// TIA Portal V17 export
// export: Created 2025-03-07T09:23:44.7208166Z, ExportSetting WithDefaults, DisplayName Totally Integrated Automation Portal, DisplayVersion V17 Update 8, DisplayName TIA Portal Openness, DisplayVersion V17 Update 8, DisplayName TIA Portal Version Control Interface, DisplayVersion V17, DisplayName SINAMICS Startdrive Advanced, DisplayVersion V17 SP2, DisplayName SINAMICS Startdrive G110M, G120, G120C, G120D, G120P, G115D, DisplayVersion V17 SP2, DisplayName SINAMICS Startdrive G130, G150, S120, S150, SINAMICS MV, S210, DisplayVersion V17 SP2, DisplayName STEP 7 Professional, DisplayVersion V17 Update 8, DisplayName SINUMERIK ONE STEP 7 Toolbox, DisplayVersion V17 Update 12, DisplayName SINUMERIK 840D sl STEP 7 Toolbox, DisplayVersion V17 Update 12, DisplayName STEP 7 Safety, DisplayVersion V17 Update 6, DisplayName WinCC Advanced, DisplayVersion V17 Update 8
FUNCTION "FC7238_VARIABLES_PLC_CONNECTION" : Void   // FC7238, LAD
{ S7_Optimized_Access := 'TRUE' }
VERSION : 0.1
// stored: AutoNumber false, IsIECCheckEnabled false, SetENOAutomatically false, UDAEnableTagReadback false
   VAR_TEMP
      AUX : Bool;
   END_VAR
   VAR_TEMP   // added for the SCL form of the ladder/FBD networks
      _w1 : Bool;
   END_VAR
BEGIN

REGION Network 1: FEEDERS GAS CHANGE CONDITIONS
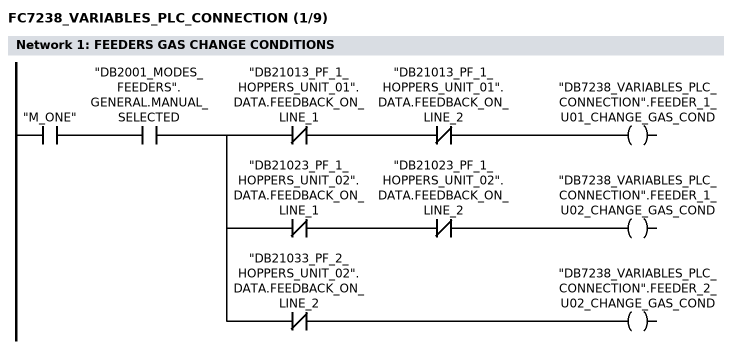
   RUNG wire#powerrail
      Contact( "M_ONE" )
      Contact( "DB2001_MODES_FEEDERS".GENERAL.MANUAL_SELECTED )
      wire#w1
      I_Contact( "DB21013_PF_1_HOPPERS_UNIT_01".DATA.FEEDBACK_ON_LINE_1 )
      I_Contact( "DB21013_PF_1_HOPPERS_UNIT_01".DATA.FEEDBACK_ON_LINE_2 )
      Coil( "DB7238_VARIABLES_PLC_CONNECTION".FEEDER_1_U01_CHANGE_GAS_COND )
   END_RUNG
   RUNG wire#w1
      I_Contact( "DB21023_PF_1_HOPPERS_UNIT_02".DATA.FEEDBACK_ON_LINE_1 )
      I_Contact( "DB21023_PF_1_HOPPERS_UNIT_02".DATA.FEEDBACK_ON_LINE_2 )
      Coil( "DB7238_VARIABLES_PLC_CONNECTION".FEEDER_1_U02_CHANGE_GAS_COND )
   END_RUNG
   RUNG wire#w1
      I_Contact( "DB21033_PF_2_HOPPERS_UNIT_02".DATA.FEEDBACK_ON_LINE_2 )
      Coil( "DB7238_VARIABLES_PLC_CONNECTION".FEEDER_2_U02_CHANGE_GAS_COND )
   END_RUNG
   // the same network as SCL:
   #_w1 := "M_ONE" AND "DB2001_MODES_FEEDERS".GENERAL.MANUAL_SELECTED;
   "DB7238_VARIABLES_PLC_CONNECTION".FEEDER_1_U01_CHANGE_GAS_COND := #_w1 AND NOT "DB21013_PF_1_HOPPERS_UNIT_01".DATA.FEEDBACK_ON_LINE_1 AND NOT "DB21013_PF_1_HOPPERS_UNIT_01".DATA.FEEDBACK_ON_LINE_2;
   "DB7238_VARIABLES_PLC_CONNECTION".FEEDER_1_U02_CHANGE_GAS_COND := #_w1 AND NOT "DB21023_PF_1_HOPPERS_UNIT_02".DATA.FEEDBACK_ON_LINE_1 AND NOT "DB21023_PF_1_HOPPERS_UNIT_02".DATA.FEEDBACK_ON_LINE_2;
   "DB7238_VARIABLES_PLC_CONNECTION".FEEDER_2_U02_CHANGE_GAS_COND := #_w1 AND NOT "DB21033_PF_2_HOPPERS_UNIT_02".DATA.FEEDBACK_ON_LINE_2;
END_REGION

REGION Network 2: FEEDER 1 UNIT 01 LINE 1
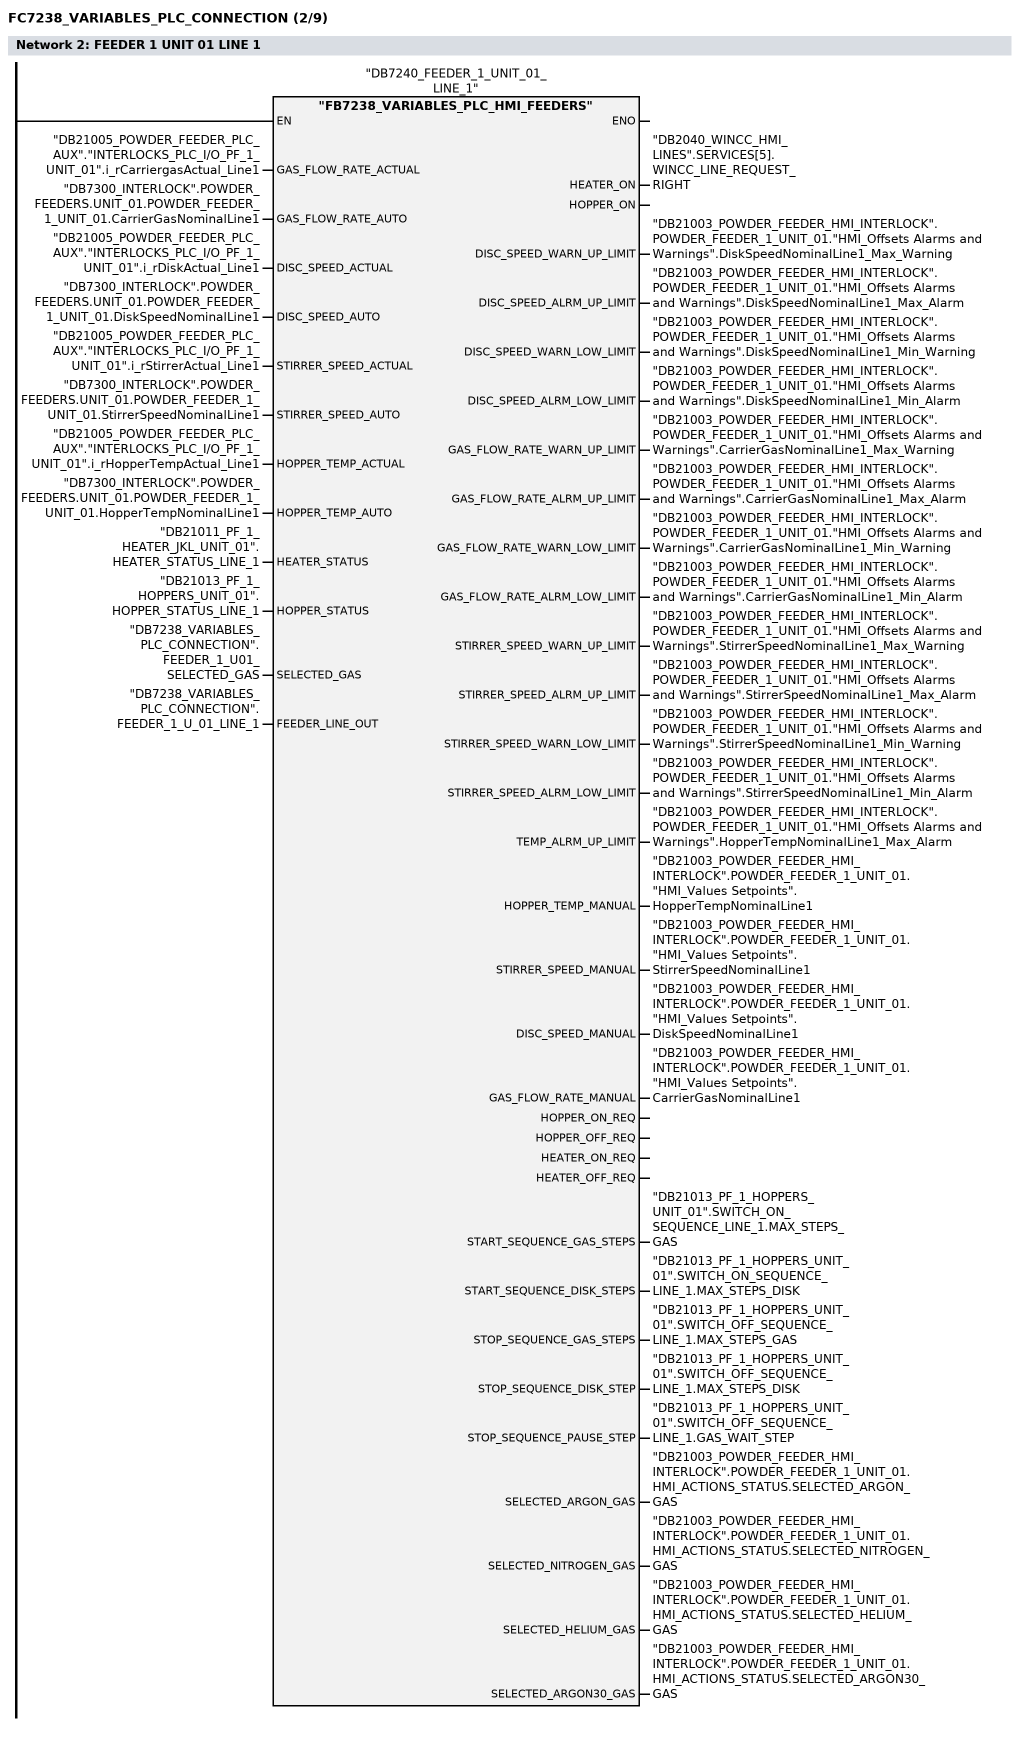
   RUNG wire#powerrail
      "DB7240_FEEDER_1_UNIT_01_LINE_1"(GAS_FLOW_RATE_ACTUAL := "DB21005_POWDER_FEEDER_PLC_AUX"."INTERLOCKS_PLC_I/O_PF_1_UNIT_01".i_rCarriergasActual_Line1, GAS_FLOW_RATE_AUTO := "DB7300_INTERLOCK".POWDER_FEEDERS.UNIT_01.POWDER_FEEDER_1_UNIT_01.CarrierGasNominalLine1, DISC_SPEED_ACTUAL := "DB21005_POWDER_FEEDER_PLC_AUX"."INTERLOCKS_PLC_I/O_PF_1_UNIT_01".i_rDiskActual_Line1, DISC_SPEED_AUTO := "DB7300_INTERLOCK".POWDER_FEEDERS.UNIT_01.POWDER_FEEDER_1_UNIT_01.DiskSpeedNominalLine1, STIRRER_SPEED_ACTUAL := "DB21005_POWDER_FEEDER_PLC_AUX"."INTERLOCKS_PLC_I/O_PF_1_UNIT_01".i_rStirrerActual_Line1, STIRRER_SPEED_AUTO := "DB7300_INTERLOCK".POWDER_FEEDERS.UNIT_01.POWDER_FEEDER_1_UNIT_01.StirrerSpeedNominalLine1, HOPPER_TEMP_ACTUAL := "DB21005_POWDER_FEEDER_PLC_AUX"."INTERLOCKS_PLC_I/O_PF_1_UNIT_01".i_rHopperTempActual_Line1, HOPPER_TEMP_AUTO := "DB7300_INTERLOCK".POWDER_FEEDERS.UNIT_01.POWDER_FEEDER_1_UNIT_01.HopperTempNominalLine1, HEATER_STATUS := "DB21011_PF_1_HEATER_JKL_UNIT_01".HEATER_STATUS_LINE_1, HOPPER_STATUS := "DB21013_PF_1_HOPPERS_UNIT_01".HOPPER_STATUS_LINE_1, SELECTED_GAS := "DB7238_VARIABLES_PLC_CONNECTION".FEEDER_1_U01_SELECTED_GAS, FEEDER_LINE_OUT := "DB7238_VARIABLES_PLC_CONNECTION".FEEDER_1_U_01_LINE_1, HEATER_ON => "DB2040_WINCC_HMI_LINES".SERVICES[5].WINCC_LINE_REQUEST_RIGHT, HOPPER_ON =>, DISC_SPEED_WARN_UP_LIMIT => "DB21003_POWDER_FEEDER_HMI_INTERLOCK".POWDER_FEEDER_1_UNIT_01."HMI_Offsets Alarms and Warnings".DiskSpeedNominalLine1_Max_Warning, DISC_SPEED_ALRM_UP_LIMIT => "DB21003_POWDER_FEEDER_HMI_INTERLOCK".POWDER_FEEDER_1_UNIT_01."HMI_Offsets Alarms and Warnings".DiskSpeedNominalLine1_Max_Alarm, DISC_SPEED_WARN_LOW_LIMIT => "DB21003_POWDER_FEEDER_HMI_INTERLOCK".POWDER_FEEDER_1_UNIT_01."HMI_Offsets Alarms and Warnings".DiskSpeedNominalLine1_Min_Warning, DISC_SPEED_ALRM_LOW_LIMIT => "DB21003_POWDER_FEEDER_HMI_INTERLOCK".POWDER_FEEDER_1_UNIT_01."HMI_Offsets Alarms and Warnings".DiskSpeedNominalLine1_Min_Alarm, GAS_FLOW_RATE_WARN_UP_LIMIT => "DB21003_POWDER_FEEDER_HMI_INTERLOCK".POWDER_FEEDER_1_UNIT_01."HMI_Offsets Alarms and Warnings".CarrierGasNominalLine1_Max_Warning, GAS_FLOW_RATE_ALRM_UP_LIMIT => "DB21003_POWDER_FEEDER_HMI_INTERLOCK".POWDER_FEEDER_1_UNIT_01."HMI_Offsets Alarms and Warnings".CarrierGasNominalLine1_Max_Alarm, GAS_FLOW_RATE_WARN_LOW_LIMIT => "DB21003_POWDER_FEEDER_HMI_INTERLOCK".POWDER_FEEDER_1_UNIT_01."HMI_Offsets Alarms and Warnings".CarrierGasNominalLine1_Min_Warning, GAS_FLOW_RATE_ALRM_LOW_LIMIT => "DB21003_POWDER_FEEDER_HMI_INTERLOCK".POWDER_FEEDER_1_UNIT_01."HMI_Offsets Alarms and Warnings".CarrierGasNominalLine1_Min_Alarm, STIRRER_SPEED_WARN_UP_LIMIT => "DB21003_POWDER_FEEDER_HMI_INTERLOCK".POWDER_FEEDER_1_UNIT_01."HMI_Offsets Alarms and Warnings".StirrerSpeedNominalLine1_Max_Warning, STIRRER_SPEED_ALRM_UP_LIMIT => "DB21003_POWDER_FEEDER_HMI_INTERLOCK".POWDER_FEEDER_1_UNIT_01."HMI_Offsets Alarms and Warnings".StirrerSpeedNominalLine1_Max_Alarm, STIRRER_SPEED_WARN_LOW_LIMIT => "DB21003_POWDER_FEEDER_HMI_INTERLOCK".POWDER_FEEDER_1_UNIT_01."HMI_Offsets Alarms and Warnings".StirrerSpeedNominalLine1_Min_Warning, STIRRER_SPEED_ALRM_LOW_LIMIT => "DB21003_POWDER_FEEDER_HMI_INTERLOCK".POWDER_FEEDER_1_UNIT_01."HMI_Offsets Alarms and Warnings".StirrerSpeedNominalLine1_Min_Alarm, TEMP_ALRM_UP_LIMIT => "DB21003_POWDER_FEEDER_HMI_INTERLOCK".POWDER_FEEDER_1_UNIT_01."HMI_Offsets Alarms and Warnings".HopperTempNominalLine1_Max_Alarm, HOPPER_TEMP_MANUAL => "DB21003_POWDER_FEEDER_HMI_INTERLOCK".POWDER_FEEDER_1_UNIT_01."HMI_Values Setpoints".HopperTempNominalLine1, STIRRER_SPEED_MANUAL => "DB21003_POWDER_FEEDER_HMI_INTERLOCK".POWDER_FEEDER_1_UNIT_01."HMI_Values Setpoints".StirrerSpeedNominalLine1, DISC_SPEED_MANUAL => "DB21003_POWDER_FEEDER_HMI_INTERLOCK".POWDER_FEEDER_1_UNIT_01."HMI_Values Setpoints".DiskSpeedNominalLine1, GAS_FLOW_RATE_MANUAL => "DB21003_POWDER_FEEDER_HMI_INTERLOCK".POWDER_FEEDER_1_UNIT_01."HMI_Values Setpoints".CarrierGasNominalLine1, HOPPER_ON_REQ =>, HOPPER_OFF_REQ =>, HEATER_ON_REQ =>, HEATER_OFF_REQ =>, START_SEQUENCE_GAS_STEPS => "DB21013_PF_1_HOPPERS_UNIT_01".SWITCH_ON_SEQUENCE_LINE_1.MAX_STEPS_GAS, START_SEQUENCE_DISK_STEPS => "DB21013_PF_1_HOPPERS_UNIT_01".SWITCH_ON_SEQUENCE_LINE_1.MAX_STEPS_DISK, STOP_SEQUENCE_GAS_STEPS => "DB21013_PF_1_HOPPERS_UNIT_01".SWITCH_OFF_SEQUENCE_LINE_1.MAX_STEPS_GAS, STOP_SEQUENCE_DISK_STEP => "DB21013_PF_1_HOPPERS_UNIT_01".SWITCH_OFF_SEQUENCE_LINE_1.MAX_STEPS_DISK, STOP_SEQUENCE_PAUSE_STEP => "DB21013_PF_1_HOPPERS_UNIT_01".SWITCH_OFF_SEQUENCE_LINE_1.GAS_WAIT_STEP, SELECTED_ARGON_GAS => "DB21003_POWDER_FEEDER_HMI_INTERLOCK".POWDER_FEEDER_1_UNIT_01.HMI_ACTIONS_STATUS.SELECTED_ARGON_GAS, SELECTED_NITROGEN_GAS => "DB21003_POWDER_FEEDER_HMI_INTERLOCK".POWDER_FEEDER_1_UNIT_01.HMI_ACTIONS_STATUS.SELECTED_NITROGEN_GAS, SELECTED_HELIUM_GAS => "DB21003_POWDER_FEEDER_HMI_INTERLOCK".POWDER_FEEDER_1_UNIT_01.HMI_ACTIONS_STATUS.SELECTED_HELIUM_GAS, SELECTED_ARGON30_GAS => "DB21003_POWDER_FEEDER_HMI_INTERLOCK".POWDER_FEEDER_1_UNIT_01.HMI_ACTIONS_STATUS.SELECTED_ARGON30_GAS)
   END_RUNG
   // the same network as SCL:
   "DB7240_FEEDER_1_UNIT_01_LINE_1"(GAS_FLOW_RATE_ACTUAL := "DB21005_POWDER_FEEDER_PLC_AUX"."INTERLOCKS_PLC_I/O_PF_1_UNIT_01".i_rCarriergasActual_Line1,   // "FB7238_VARIABLES_PLC_HMI_FEEDERS"
                           GAS_FLOW_RATE_AUTO := "DB7300_INTERLOCK".POWDER_FEEDERS.UNIT_01.POWDER_FEEDER_1_UNIT_01.CarrierGasNominalLine1,
                           DISC_SPEED_ACTUAL := "DB21005_POWDER_FEEDER_PLC_AUX"."INTERLOCKS_PLC_I/O_PF_1_UNIT_01".i_rDiskActual_Line1,
                           DISC_SPEED_AUTO := "DB7300_INTERLOCK".POWDER_FEEDERS.UNIT_01.POWDER_FEEDER_1_UNIT_01.DiskSpeedNominalLine1,
                           STIRRER_SPEED_ACTUAL := "DB21005_POWDER_FEEDER_PLC_AUX"."INTERLOCKS_PLC_I/O_PF_1_UNIT_01".i_rStirrerActual_Line1,
                           STIRRER_SPEED_AUTO := "DB7300_INTERLOCK".POWDER_FEEDERS.UNIT_01.POWDER_FEEDER_1_UNIT_01.StirrerSpeedNominalLine1,
                           HOPPER_TEMP_ACTUAL := "DB21005_POWDER_FEEDER_PLC_AUX"."INTERLOCKS_PLC_I/O_PF_1_UNIT_01".i_rHopperTempActual_Line1,
                           HOPPER_TEMP_AUTO := "DB7300_INTERLOCK".POWDER_FEEDERS.UNIT_01.POWDER_FEEDER_1_UNIT_01.HopperTempNominalLine1,
                           HEATER_STATUS := "DB21011_PF_1_HEATER_JKL_UNIT_01".HEATER_STATUS_LINE_1,
                           HOPPER_STATUS := "DB21013_PF_1_HOPPERS_UNIT_01".HOPPER_STATUS_LINE_1,
                           SELECTED_GAS := "DB7238_VARIABLES_PLC_CONNECTION".FEEDER_1_U01_SELECTED_GAS,
                           FEEDER_LINE_OUT := "DB7238_VARIABLES_PLC_CONNECTION".FEEDER_1_U_01_LINE_1,
                           HEATER_ON => "DB2040_WINCC_HMI_LINES".SERVICES[5].WINCC_LINE_REQUEST_RIGHT,
                           DISC_SPEED_WARN_UP_LIMIT => "DB21003_POWDER_FEEDER_HMI_INTERLOCK".POWDER_FEEDER_1_UNIT_01."HMI_Offsets Alarms and Warnings".DiskSpeedNominalLine1_Max_Warning,
                           DISC_SPEED_ALRM_UP_LIMIT => "DB21003_POWDER_FEEDER_HMI_INTERLOCK".POWDER_FEEDER_1_UNIT_01."HMI_Offsets Alarms and Warnings".DiskSpeedNominalLine1_Max_Alarm,
                           DISC_SPEED_WARN_LOW_LIMIT => "DB21003_POWDER_FEEDER_HMI_INTERLOCK".POWDER_FEEDER_1_UNIT_01."HMI_Offsets Alarms and Warnings".DiskSpeedNominalLine1_Min_Warning,
                           DISC_SPEED_ALRM_LOW_LIMIT => "DB21003_POWDER_FEEDER_HMI_INTERLOCK".POWDER_FEEDER_1_UNIT_01."HMI_Offsets Alarms and Warnings".DiskSpeedNominalLine1_Min_Alarm,
                           GAS_FLOW_RATE_WARN_UP_LIMIT => "DB21003_POWDER_FEEDER_HMI_INTERLOCK".POWDER_FEEDER_1_UNIT_01."HMI_Offsets Alarms and Warnings".CarrierGasNominalLine1_Max_Warning,
                           GAS_FLOW_RATE_ALRM_UP_LIMIT => "DB21003_POWDER_FEEDER_HMI_INTERLOCK".POWDER_FEEDER_1_UNIT_01."HMI_Offsets Alarms and Warnings".CarrierGasNominalLine1_Max_Alarm,
                           GAS_FLOW_RATE_WARN_LOW_LIMIT => "DB21003_POWDER_FEEDER_HMI_INTERLOCK".POWDER_FEEDER_1_UNIT_01."HMI_Offsets Alarms and Warnings".CarrierGasNominalLine1_Min_Warning,
                           GAS_FLOW_RATE_ALRM_LOW_LIMIT => "DB21003_POWDER_FEEDER_HMI_INTERLOCK".POWDER_FEEDER_1_UNIT_01."HMI_Offsets Alarms and Warnings".CarrierGasNominalLine1_Min_Alarm,
                           STIRRER_SPEED_WARN_UP_LIMIT => "DB21003_POWDER_FEEDER_HMI_INTERLOCK".POWDER_FEEDER_1_UNIT_01."HMI_Offsets Alarms and Warnings".StirrerSpeedNominalLine1_Max_Warning,
                           STIRRER_SPEED_ALRM_UP_LIMIT => "DB21003_POWDER_FEEDER_HMI_INTERLOCK".POWDER_FEEDER_1_UNIT_01."HMI_Offsets Alarms and Warnings".StirrerSpeedNominalLine1_Max_Alarm,
                           STIRRER_SPEED_WARN_LOW_LIMIT => "DB21003_POWDER_FEEDER_HMI_INTERLOCK".POWDER_FEEDER_1_UNIT_01."HMI_Offsets Alarms and Warnings".StirrerSpeedNominalLine1_Min_Warning,
                           STIRRER_SPEED_ALRM_LOW_LIMIT => "DB21003_POWDER_FEEDER_HMI_INTERLOCK".POWDER_FEEDER_1_UNIT_01."HMI_Offsets Alarms and Warnings".StirrerSpeedNominalLine1_Min_Alarm,
                           TEMP_ALRM_UP_LIMIT => "DB21003_POWDER_FEEDER_HMI_INTERLOCK".POWDER_FEEDER_1_UNIT_01."HMI_Offsets Alarms and Warnings".HopperTempNominalLine1_Max_Alarm,
                           HOPPER_TEMP_MANUAL => "DB21003_POWDER_FEEDER_HMI_INTERLOCK".POWDER_FEEDER_1_UNIT_01."HMI_Values Setpoints".HopperTempNominalLine1,
                           STIRRER_SPEED_MANUAL => "DB21003_POWDER_FEEDER_HMI_INTERLOCK".POWDER_FEEDER_1_UNIT_01."HMI_Values Setpoints".StirrerSpeedNominalLine1,
                           DISC_SPEED_MANUAL => "DB21003_POWDER_FEEDER_HMI_INTERLOCK".POWDER_FEEDER_1_UNIT_01."HMI_Values Setpoints".DiskSpeedNominalLine1,
                           GAS_FLOW_RATE_MANUAL => "DB21003_POWDER_FEEDER_HMI_INTERLOCK".POWDER_FEEDER_1_UNIT_01."HMI_Values Setpoints".CarrierGasNominalLine1,
                           START_SEQUENCE_GAS_STEPS => "DB21013_PF_1_HOPPERS_UNIT_01".SWITCH_ON_SEQUENCE_LINE_1.MAX_STEPS_GAS,
                           START_SEQUENCE_DISK_STEPS => "DB21013_PF_1_HOPPERS_UNIT_01".SWITCH_ON_SEQUENCE_LINE_1.MAX_STEPS_DISK,
                           STOP_SEQUENCE_GAS_STEPS => "DB21013_PF_1_HOPPERS_UNIT_01".SWITCH_OFF_SEQUENCE_LINE_1.MAX_STEPS_GAS,
                           STOP_SEQUENCE_DISK_STEP => "DB21013_PF_1_HOPPERS_UNIT_01".SWITCH_OFF_SEQUENCE_LINE_1.MAX_STEPS_DISK,
                           STOP_SEQUENCE_PAUSE_STEP => "DB21013_PF_1_HOPPERS_UNIT_01".SWITCH_OFF_SEQUENCE_LINE_1.GAS_WAIT_STEP,
                           SELECTED_ARGON_GAS => "DB21003_POWDER_FEEDER_HMI_INTERLOCK".POWDER_FEEDER_1_UNIT_01.HMI_ACTIONS_STATUS.SELECTED_ARGON_GAS,
                           SELECTED_NITROGEN_GAS => "DB21003_POWDER_FEEDER_HMI_INTERLOCK".POWDER_FEEDER_1_UNIT_01.HMI_ACTIONS_STATUS.SELECTED_NITROGEN_GAS,
                           SELECTED_HELIUM_GAS => "DB21003_POWDER_FEEDER_HMI_INTERLOCK".POWDER_FEEDER_1_UNIT_01.HMI_ACTIONS_STATUS.SELECTED_HELIUM_GAS,
                           SELECTED_ARGON30_GAS => "DB21003_POWDER_FEEDER_HMI_INTERLOCK".POWDER_FEEDER_1_UNIT_01.HMI_ACTIONS_STATUS.SELECTED_ARGON30_GAS);
END_REGION

REGION Network 3: FEEDER 1 UNIT 01 LINE 2
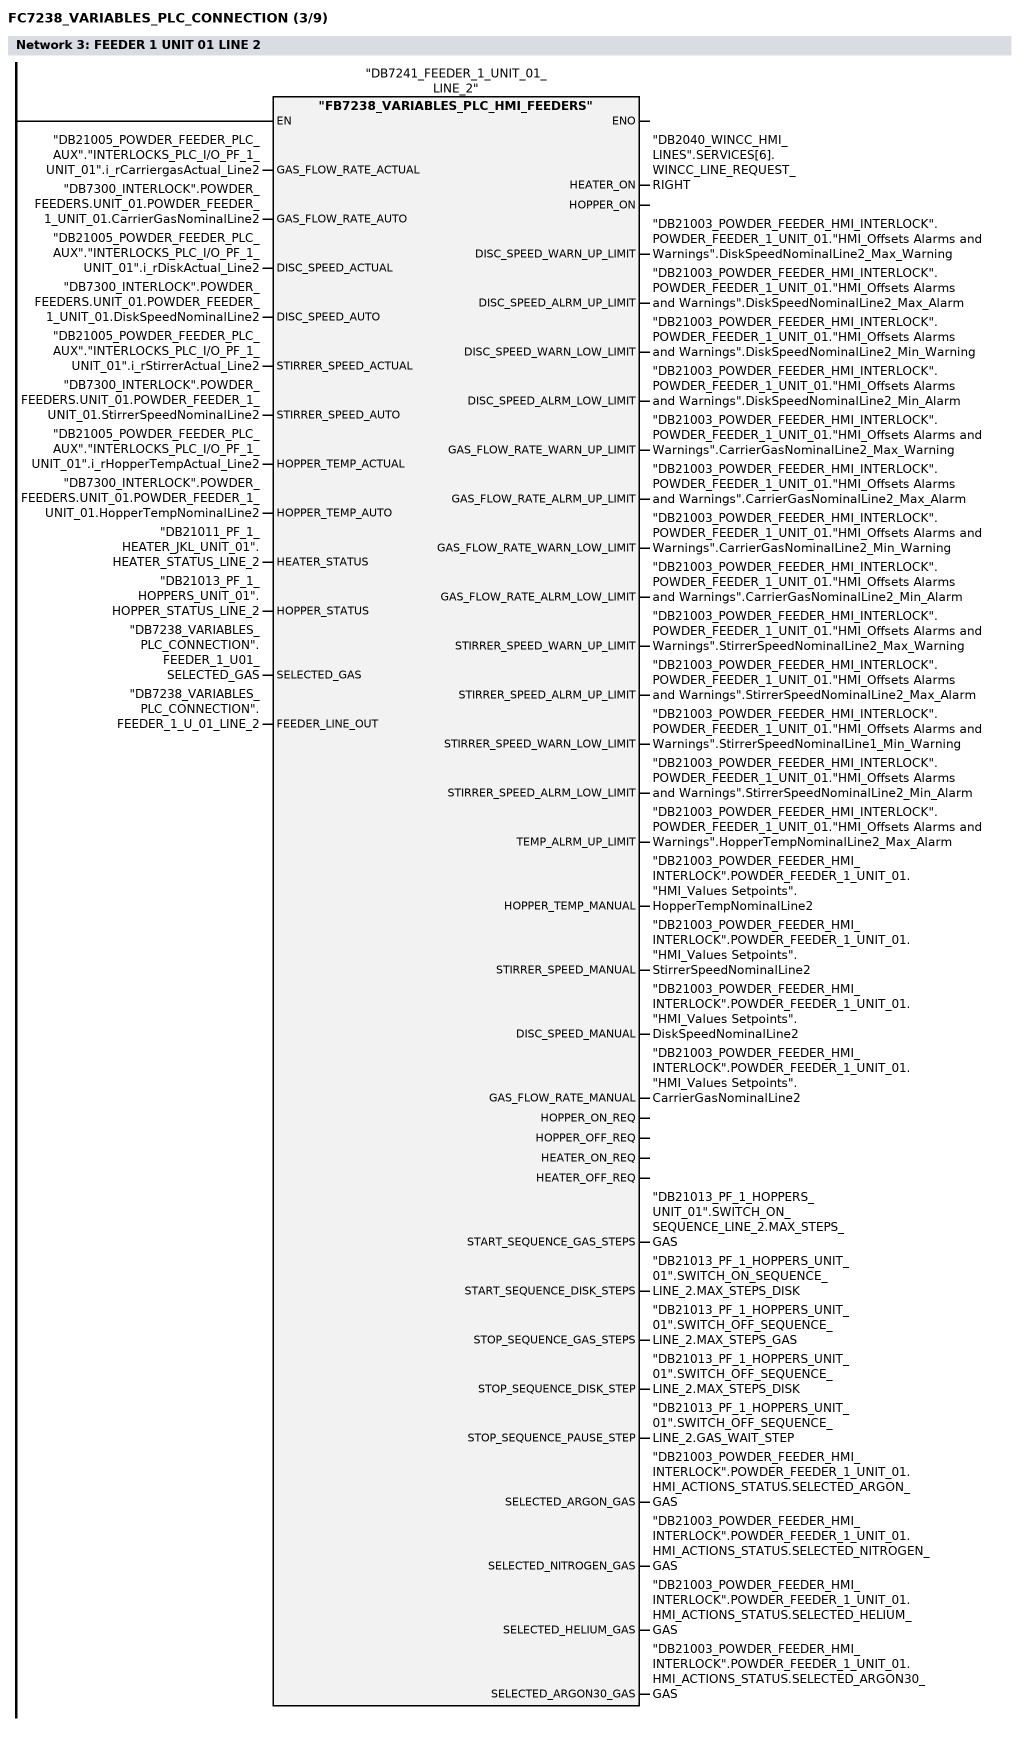
   RUNG wire#powerrail
      "DB7241_FEEDER_1_UNIT_01_LINE_2"(GAS_FLOW_RATE_ACTUAL := "DB21005_POWDER_FEEDER_PLC_AUX"."INTERLOCKS_PLC_I/O_PF_1_UNIT_01".i_rCarriergasActual_Line2, GAS_FLOW_RATE_AUTO := "DB7300_INTERLOCK".POWDER_FEEDERS.UNIT_01.POWDER_FEEDER_1_UNIT_01.CarrierGasNominalLine2, DISC_SPEED_ACTUAL := "DB21005_POWDER_FEEDER_PLC_AUX"."INTERLOCKS_PLC_I/O_PF_1_UNIT_01".i_rDiskActual_Line2, DISC_SPEED_AUTO := "DB7300_INTERLOCK".POWDER_FEEDERS.UNIT_01.POWDER_FEEDER_1_UNIT_01.DiskSpeedNominalLine2, STIRRER_SPEED_ACTUAL := "DB21005_POWDER_FEEDER_PLC_AUX"."INTERLOCKS_PLC_I/O_PF_1_UNIT_01".i_rStirrerActual_Line2, STIRRER_SPEED_AUTO := "DB7300_INTERLOCK".POWDER_FEEDERS.UNIT_01.POWDER_FEEDER_1_UNIT_01.StirrerSpeedNominalLine2, HOPPER_TEMP_ACTUAL := "DB21005_POWDER_FEEDER_PLC_AUX"."INTERLOCKS_PLC_I/O_PF_1_UNIT_01".i_rHopperTempActual_Line2, HOPPER_TEMP_AUTO := "DB7300_INTERLOCK".POWDER_FEEDERS.UNIT_01.POWDER_FEEDER_1_UNIT_01.HopperTempNominalLine2, HEATER_STATUS := "DB21011_PF_1_HEATER_JKL_UNIT_01".HEATER_STATUS_LINE_2, HOPPER_STATUS := "DB21013_PF_1_HOPPERS_UNIT_01".HOPPER_STATUS_LINE_2, SELECTED_GAS := "DB7238_VARIABLES_PLC_CONNECTION".FEEDER_1_U01_SELECTED_GAS, FEEDER_LINE_OUT := "DB7238_VARIABLES_PLC_CONNECTION".FEEDER_1_U_01_LINE_2, HEATER_ON => "DB2040_WINCC_HMI_LINES".SERVICES[6].WINCC_LINE_REQUEST_RIGHT, HOPPER_ON =>, DISC_SPEED_WARN_UP_LIMIT => "DB21003_POWDER_FEEDER_HMI_INTERLOCK".POWDER_FEEDER_1_UNIT_01."HMI_Offsets Alarms and Warnings".DiskSpeedNominalLine2_Max_Warning, DISC_SPEED_ALRM_UP_LIMIT => "DB21003_POWDER_FEEDER_HMI_INTERLOCK".POWDER_FEEDER_1_UNIT_01."HMI_Offsets Alarms and Warnings".DiskSpeedNominalLine2_Max_Alarm, DISC_SPEED_WARN_LOW_LIMIT => "DB21003_POWDER_FEEDER_HMI_INTERLOCK".POWDER_FEEDER_1_UNIT_01."HMI_Offsets Alarms and Warnings".DiskSpeedNominalLine2_Min_Warning, DISC_SPEED_ALRM_LOW_LIMIT => "DB21003_POWDER_FEEDER_HMI_INTERLOCK".POWDER_FEEDER_1_UNIT_01."HMI_Offsets Alarms and Warnings".DiskSpeedNominalLine2_Min_Alarm, GAS_FLOW_RATE_WARN_UP_LIMIT => "DB21003_POWDER_FEEDER_HMI_INTERLOCK".POWDER_FEEDER_1_UNIT_01."HMI_Offsets Alarms and Warnings".CarrierGasNominalLine2_Max_Warning, GAS_FLOW_RATE_ALRM_UP_LIMIT => "DB21003_POWDER_FEEDER_HMI_INTERLOCK".POWDER_FEEDER_1_UNIT_01."HMI_Offsets Alarms and Warnings".CarrierGasNominalLine2_Max_Alarm, GAS_FLOW_RATE_WARN_LOW_LIMIT => "DB21003_POWDER_FEEDER_HMI_INTERLOCK".POWDER_FEEDER_1_UNIT_01."HMI_Offsets Alarms and Warnings".CarrierGasNominalLine2_Min_Warning, GAS_FLOW_RATE_ALRM_LOW_LIMIT => "DB21003_POWDER_FEEDER_HMI_INTERLOCK".POWDER_FEEDER_1_UNIT_01."HMI_Offsets Alarms and Warnings".CarrierGasNominalLine2_Min_Alarm, STIRRER_SPEED_WARN_UP_LIMIT => "DB21003_POWDER_FEEDER_HMI_INTERLOCK".POWDER_FEEDER_1_UNIT_01."HMI_Offsets Alarms and Warnings".StirrerSpeedNominalLine2_Max_Warning, STIRRER_SPEED_ALRM_UP_LIMIT => "DB21003_POWDER_FEEDER_HMI_INTERLOCK".POWDER_FEEDER_1_UNIT_01."HMI_Offsets Alarms and Warnings".StirrerSpeedNominalLine2_Max_Alarm, STIRRER_SPEED_WARN_LOW_LIMIT => "DB21003_POWDER_FEEDER_HMI_INTERLOCK".POWDER_FEEDER_1_UNIT_01."HMI_Offsets Alarms and Warnings".StirrerSpeedNominalLine1_Min_Warning, STIRRER_SPEED_ALRM_LOW_LIMIT => "DB21003_POWDER_FEEDER_HMI_INTERLOCK".POWDER_FEEDER_1_UNIT_01."HMI_Offsets Alarms and Warnings".StirrerSpeedNominalLine2_Min_Alarm, TEMP_ALRM_UP_LIMIT => "DB21003_POWDER_FEEDER_HMI_INTERLOCK".POWDER_FEEDER_1_UNIT_01."HMI_Offsets Alarms and Warnings".HopperTempNominalLine2_Max_Alarm, HOPPER_TEMP_MANUAL => "DB21003_POWDER_FEEDER_HMI_INTERLOCK".POWDER_FEEDER_1_UNIT_01."HMI_Values Setpoints".HopperTempNominalLine2, STIRRER_SPEED_MANUAL => "DB21003_POWDER_FEEDER_HMI_INTERLOCK".POWDER_FEEDER_1_UNIT_01."HMI_Values Setpoints".StirrerSpeedNominalLine2, DISC_SPEED_MANUAL => "DB21003_POWDER_FEEDER_HMI_INTERLOCK".POWDER_FEEDER_1_UNIT_01."HMI_Values Setpoints".DiskSpeedNominalLine2, GAS_FLOW_RATE_MANUAL => "DB21003_POWDER_FEEDER_HMI_INTERLOCK".POWDER_FEEDER_1_UNIT_01."HMI_Values Setpoints".CarrierGasNominalLine2, HOPPER_ON_REQ =>, HOPPER_OFF_REQ =>, HEATER_ON_REQ =>, HEATER_OFF_REQ =>, START_SEQUENCE_GAS_STEPS => "DB21013_PF_1_HOPPERS_UNIT_01".SWITCH_ON_SEQUENCE_LINE_2.MAX_STEPS_GAS, START_SEQUENCE_DISK_STEPS => "DB21013_PF_1_HOPPERS_UNIT_01".SWITCH_ON_SEQUENCE_LINE_2.MAX_STEPS_DISK, STOP_SEQUENCE_GAS_STEPS => "DB21013_PF_1_HOPPERS_UNIT_01".SWITCH_OFF_SEQUENCE_LINE_2.MAX_STEPS_GAS, STOP_SEQUENCE_DISK_STEP => "DB21013_PF_1_HOPPERS_UNIT_01".SWITCH_OFF_SEQUENCE_LINE_2.MAX_STEPS_DISK, STOP_SEQUENCE_PAUSE_STEP => "DB21013_PF_1_HOPPERS_UNIT_01".SWITCH_OFF_SEQUENCE_LINE_2.GAS_WAIT_STEP, SELECTED_ARGON_GAS => "DB21003_POWDER_FEEDER_HMI_INTERLOCK".POWDER_FEEDER_1_UNIT_01.HMI_ACTIONS_STATUS.SELECTED_ARGON_GAS, SELECTED_NITROGEN_GAS => "DB21003_POWDER_FEEDER_HMI_INTERLOCK".POWDER_FEEDER_1_UNIT_01.HMI_ACTIONS_STATUS.SELECTED_NITROGEN_GAS, SELECTED_HELIUM_GAS => "DB21003_POWDER_FEEDER_HMI_INTERLOCK".POWDER_FEEDER_1_UNIT_01.HMI_ACTIONS_STATUS.SELECTED_HELIUM_GAS, SELECTED_ARGON30_GAS => "DB21003_POWDER_FEEDER_HMI_INTERLOCK".POWDER_FEEDER_1_UNIT_01.HMI_ACTIONS_STATUS.SELECTED_ARGON30_GAS)
   END_RUNG
   // the same network as SCL:
   "DB7241_FEEDER_1_UNIT_01_LINE_2"(GAS_FLOW_RATE_ACTUAL := "DB21005_POWDER_FEEDER_PLC_AUX"."INTERLOCKS_PLC_I/O_PF_1_UNIT_01".i_rCarriergasActual_Line2,   // "FB7238_VARIABLES_PLC_HMI_FEEDERS"
                           GAS_FLOW_RATE_AUTO := "DB7300_INTERLOCK".POWDER_FEEDERS.UNIT_01.POWDER_FEEDER_1_UNIT_01.CarrierGasNominalLine2,
                           DISC_SPEED_ACTUAL := "DB21005_POWDER_FEEDER_PLC_AUX"."INTERLOCKS_PLC_I/O_PF_1_UNIT_01".i_rDiskActual_Line2,
                           DISC_SPEED_AUTO := "DB7300_INTERLOCK".POWDER_FEEDERS.UNIT_01.POWDER_FEEDER_1_UNIT_01.DiskSpeedNominalLine2,
                           STIRRER_SPEED_ACTUAL := "DB21005_POWDER_FEEDER_PLC_AUX"."INTERLOCKS_PLC_I/O_PF_1_UNIT_01".i_rStirrerActual_Line2,
                           STIRRER_SPEED_AUTO := "DB7300_INTERLOCK".POWDER_FEEDERS.UNIT_01.POWDER_FEEDER_1_UNIT_01.StirrerSpeedNominalLine2,
                           HOPPER_TEMP_ACTUAL := "DB21005_POWDER_FEEDER_PLC_AUX"."INTERLOCKS_PLC_I/O_PF_1_UNIT_01".i_rHopperTempActual_Line2,
                           HOPPER_TEMP_AUTO := "DB7300_INTERLOCK".POWDER_FEEDERS.UNIT_01.POWDER_FEEDER_1_UNIT_01.HopperTempNominalLine2,
                           HEATER_STATUS := "DB21011_PF_1_HEATER_JKL_UNIT_01".HEATER_STATUS_LINE_2,
                           HOPPER_STATUS := "DB21013_PF_1_HOPPERS_UNIT_01".HOPPER_STATUS_LINE_2,
                           SELECTED_GAS := "DB7238_VARIABLES_PLC_CONNECTION".FEEDER_1_U01_SELECTED_GAS,
                           FEEDER_LINE_OUT := "DB7238_VARIABLES_PLC_CONNECTION".FEEDER_1_U_01_LINE_2,
                           HEATER_ON => "DB2040_WINCC_HMI_LINES".SERVICES[6].WINCC_LINE_REQUEST_RIGHT,
                           DISC_SPEED_WARN_UP_LIMIT => "DB21003_POWDER_FEEDER_HMI_INTERLOCK".POWDER_FEEDER_1_UNIT_01."HMI_Offsets Alarms and Warnings".DiskSpeedNominalLine2_Max_Warning,
                           DISC_SPEED_ALRM_UP_LIMIT => "DB21003_POWDER_FEEDER_HMI_INTERLOCK".POWDER_FEEDER_1_UNIT_01."HMI_Offsets Alarms and Warnings".DiskSpeedNominalLine2_Max_Alarm,
                           DISC_SPEED_WARN_LOW_LIMIT => "DB21003_POWDER_FEEDER_HMI_INTERLOCK".POWDER_FEEDER_1_UNIT_01."HMI_Offsets Alarms and Warnings".DiskSpeedNominalLine2_Min_Warning,
                           DISC_SPEED_ALRM_LOW_LIMIT => "DB21003_POWDER_FEEDER_HMI_INTERLOCK".POWDER_FEEDER_1_UNIT_01."HMI_Offsets Alarms and Warnings".DiskSpeedNominalLine2_Min_Alarm,
                           GAS_FLOW_RATE_WARN_UP_LIMIT => "DB21003_POWDER_FEEDER_HMI_INTERLOCK".POWDER_FEEDER_1_UNIT_01."HMI_Offsets Alarms and Warnings".CarrierGasNominalLine2_Max_Warning,
                           GAS_FLOW_RATE_ALRM_UP_LIMIT => "DB21003_POWDER_FEEDER_HMI_INTERLOCK".POWDER_FEEDER_1_UNIT_01."HMI_Offsets Alarms and Warnings".CarrierGasNominalLine2_Max_Alarm,
                           GAS_FLOW_RATE_WARN_LOW_LIMIT => "DB21003_POWDER_FEEDER_HMI_INTERLOCK".POWDER_FEEDER_1_UNIT_01."HMI_Offsets Alarms and Warnings".CarrierGasNominalLine2_Min_Warning,
                           GAS_FLOW_RATE_ALRM_LOW_LIMIT => "DB21003_POWDER_FEEDER_HMI_INTERLOCK".POWDER_FEEDER_1_UNIT_01."HMI_Offsets Alarms and Warnings".CarrierGasNominalLine2_Min_Alarm,
                           STIRRER_SPEED_WARN_UP_LIMIT => "DB21003_POWDER_FEEDER_HMI_INTERLOCK".POWDER_FEEDER_1_UNIT_01."HMI_Offsets Alarms and Warnings".StirrerSpeedNominalLine2_Max_Warning,
                           STIRRER_SPEED_ALRM_UP_LIMIT => "DB21003_POWDER_FEEDER_HMI_INTERLOCK".POWDER_FEEDER_1_UNIT_01."HMI_Offsets Alarms and Warnings".StirrerSpeedNominalLine2_Max_Alarm,
                           STIRRER_SPEED_WARN_LOW_LIMIT => "DB21003_POWDER_FEEDER_HMI_INTERLOCK".POWDER_FEEDER_1_UNIT_01."HMI_Offsets Alarms and Warnings".StirrerSpeedNominalLine1_Min_Warning,
                           STIRRER_SPEED_ALRM_LOW_LIMIT => "DB21003_POWDER_FEEDER_HMI_INTERLOCK".POWDER_FEEDER_1_UNIT_01."HMI_Offsets Alarms and Warnings".StirrerSpeedNominalLine2_Min_Alarm,
                           TEMP_ALRM_UP_LIMIT => "DB21003_POWDER_FEEDER_HMI_INTERLOCK".POWDER_FEEDER_1_UNIT_01."HMI_Offsets Alarms and Warnings".HopperTempNominalLine2_Max_Alarm,
                           HOPPER_TEMP_MANUAL => "DB21003_POWDER_FEEDER_HMI_INTERLOCK".POWDER_FEEDER_1_UNIT_01."HMI_Values Setpoints".HopperTempNominalLine2,
                           STIRRER_SPEED_MANUAL => "DB21003_POWDER_FEEDER_HMI_INTERLOCK".POWDER_FEEDER_1_UNIT_01."HMI_Values Setpoints".StirrerSpeedNominalLine2,
                           DISC_SPEED_MANUAL => "DB21003_POWDER_FEEDER_HMI_INTERLOCK".POWDER_FEEDER_1_UNIT_01."HMI_Values Setpoints".DiskSpeedNominalLine2,
                           GAS_FLOW_RATE_MANUAL => "DB21003_POWDER_FEEDER_HMI_INTERLOCK".POWDER_FEEDER_1_UNIT_01."HMI_Values Setpoints".CarrierGasNominalLine2,
                           START_SEQUENCE_GAS_STEPS => "DB21013_PF_1_HOPPERS_UNIT_01".SWITCH_ON_SEQUENCE_LINE_2.MAX_STEPS_GAS,
                           START_SEQUENCE_DISK_STEPS => "DB21013_PF_1_HOPPERS_UNIT_01".SWITCH_ON_SEQUENCE_LINE_2.MAX_STEPS_DISK,
                           STOP_SEQUENCE_GAS_STEPS => "DB21013_PF_1_HOPPERS_UNIT_01".SWITCH_OFF_SEQUENCE_LINE_2.MAX_STEPS_GAS,
                           STOP_SEQUENCE_DISK_STEP => "DB21013_PF_1_HOPPERS_UNIT_01".SWITCH_OFF_SEQUENCE_LINE_2.MAX_STEPS_DISK,
                           STOP_SEQUENCE_PAUSE_STEP => "DB21013_PF_1_HOPPERS_UNIT_01".SWITCH_OFF_SEQUENCE_LINE_2.GAS_WAIT_STEP,
                           SELECTED_ARGON_GAS => "DB21003_POWDER_FEEDER_HMI_INTERLOCK".POWDER_FEEDER_1_UNIT_01.HMI_ACTIONS_STATUS.SELECTED_ARGON_GAS,
                           SELECTED_NITROGEN_GAS => "DB21003_POWDER_FEEDER_HMI_INTERLOCK".POWDER_FEEDER_1_UNIT_01.HMI_ACTIONS_STATUS.SELECTED_NITROGEN_GAS,
                           SELECTED_HELIUM_GAS => "DB21003_POWDER_FEEDER_HMI_INTERLOCK".POWDER_FEEDER_1_UNIT_01.HMI_ACTIONS_STATUS.SELECTED_HELIUM_GAS,
                           SELECTED_ARGON30_GAS => "DB21003_POWDER_FEEDER_HMI_INTERLOCK".POWDER_FEEDER_1_UNIT_01.HMI_ACTIONS_STATUS.SELECTED_ARGON30_GAS);
END_REGION

REGION Network 4: FEEDER 1 UNIT 02 LINE 1
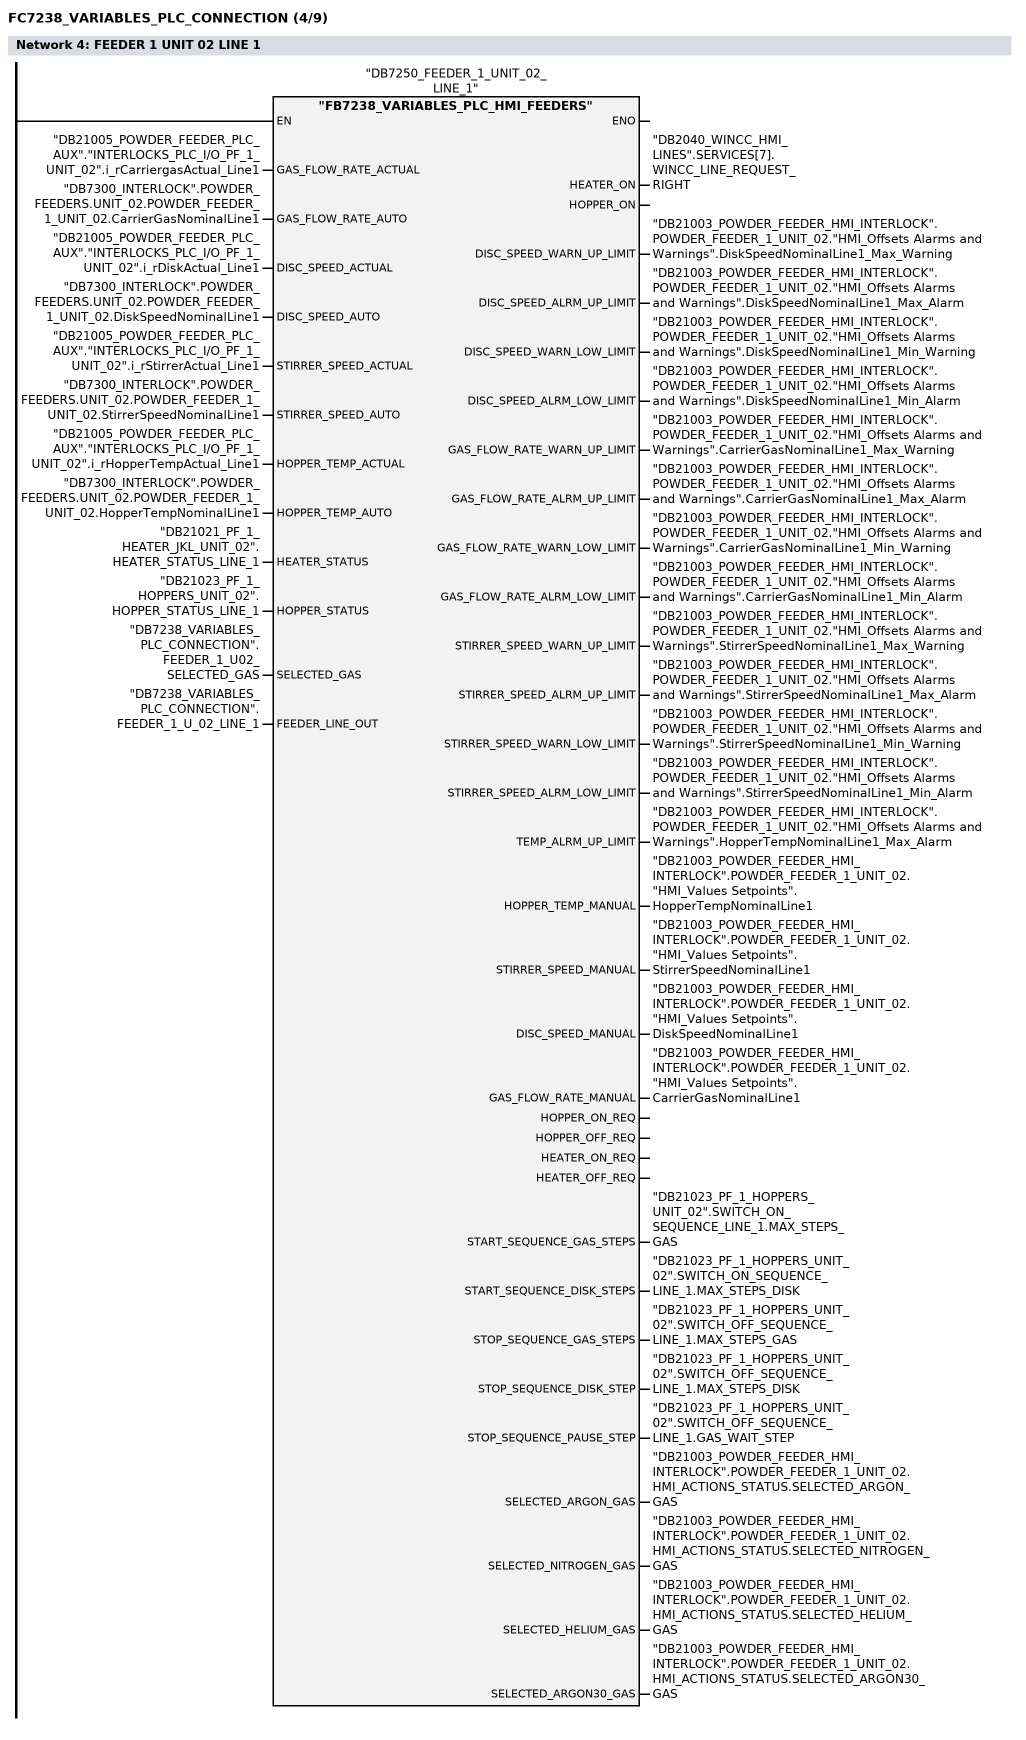
   RUNG wire#powerrail
      "DB7250_FEEDER_1_UNIT_02_LINE_1"(GAS_FLOW_RATE_ACTUAL := "DB21005_POWDER_FEEDER_PLC_AUX"."INTERLOCKS_PLC_I/O_PF_1_UNIT_02".i_rCarriergasActual_Line1, GAS_FLOW_RATE_AUTO := "DB7300_INTERLOCK".POWDER_FEEDERS.UNIT_02.POWDER_FEEDER_1_UNIT_02.CarrierGasNominalLine1, DISC_SPEED_ACTUAL := "DB21005_POWDER_FEEDER_PLC_AUX"."INTERLOCKS_PLC_I/O_PF_1_UNIT_02".i_rDiskActual_Line1, DISC_SPEED_AUTO := "DB7300_INTERLOCK".POWDER_FEEDERS.UNIT_02.POWDER_FEEDER_1_UNIT_02.DiskSpeedNominalLine1, STIRRER_SPEED_ACTUAL := "DB21005_POWDER_FEEDER_PLC_AUX"."INTERLOCKS_PLC_I/O_PF_1_UNIT_02".i_rStirrerActual_Line1, STIRRER_SPEED_AUTO := "DB7300_INTERLOCK".POWDER_FEEDERS.UNIT_02.POWDER_FEEDER_1_UNIT_02.StirrerSpeedNominalLine1, HOPPER_TEMP_ACTUAL := "DB21005_POWDER_FEEDER_PLC_AUX"."INTERLOCKS_PLC_I/O_PF_1_UNIT_02".i_rHopperTempActual_Line1, HOPPER_TEMP_AUTO := "DB7300_INTERLOCK".POWDER_FEEDERS.UNIT_02.POWDER_FEEDER_1_UNIT_02.HopperTempNominalLine1, HEATER_STATUS := "DB21021_PF_1_HEATER_JKL_UNIT_02".HEATER_STATUS_LINE_1, HOPPER_STATUS := "DB21023_PF_1_HOPPERS_UNIT_02".HOPPER_STATUS_LINE_1, SELECTED_GAS := "DB7238_VARIABLES_PLC_CONNECTION".FEEDER_1_U02_SELECTED_GAS, FEEDER_LINE_OUT := "DB7238_VARIABLES_PLC_CONNECTION".FEEDER_1_U_02_LINE_1, HEATER_ON => "DB2040_WINCC_HMI_LINES".SERVICES[7].WINCC_LINE_REQUEST_RIGHT, HOPPER_ON =>, DISC_SPEED_WARN_UP_LIMIT => "DB21003_POWDER_FEEDER_HMI_INTERLOCK".POWDER_FEEDER_1_UNIT_02."HMI_Offsets Alarms and Warnings".DiskSpeedNominalLine1_Max_Warning, DISC_SPEED_ALRM_UP_LIMIT => "DB21003_POWDER_FEEDER_HMI_INTERLOCK".POWDER_FEEDER_1_UNIT_02."HMI_Offsets Alarms and Warnings".DiskSpeedNominalLine1_Max_Alarm, DISC_SPEED_WARN_LOW_LIMIT => "DB21003_POWDER_FEEDER_HMI_INTERLOCK".POWDER_FEEDER_1_UNIT_02."HMI_Offsets Alarms and Warnings".DiskSpeedNominalLine1_Min_Warning, DISC_SPEED_ALRM_LOW_LIMIT => "DB21003_POWDER_FEEDER_HMI_INTERLOCK".POWDER_FEEDER_1_UNIT_02."HMI_Offsets Alarms and Warnings".DiskSpeedNominalLine1_Min_Alarm, GAS_FLOW_RATE_WARN_UP_LIMIT => "DB21003_POWDER_FEEDER_HMI_INTERLOCK".POWDER_FEEDER_1_UNIT_02."HMI_Offsets Alarms and Warnings".CarrierGasNominalLine1_Max_Warning, GAS_FLOW_RATE_ALRM_UP_LIMIT => "DB21003_POWDER_FEEDER_HMI_INTERLOCK".POWDER_FEEDER_1_UNIT_02."HMI_Offsets Alarms and Warnings".CarrierGasNominalLine1_Max_Alarm, GAS_FLOW_RATE_WARN_LOW_LIMIT => "DB21003_POWDER_FEEDER_HMI_INTERLOCK".POWDER_FEEDER_1_UNIT_02."HMI_Offsets Alarms and Warnings".CarrierGasNominalLine1_Min_Warning, GAS_FLOW_RATE_ALRM_LOW_LIMIT => "DB21003_POWDER_FEEDER_HMI_INTERLOCK".POWDER_FEEDER_1_UNIT_02."HMI_Offsets Alarms and Warnings".CarrierGasNominalLine1_Min_Alarm, STIRRER_SPEED_WARN_UP_LIMIT => "DB21003_POWDER_FEEDER_HMI_INTERLOCK".POWDER_FEEDER_1_UNIT_02."HMI_Offsets Alarms and Warnings".StirrerSpeedNominalLine1_Max_Warning, STIRRER_SPEED_ALRM_UP_LIMIT => "DB21003_POWDER_FEEDER_HMI_INTERLOCK".POWDER_FEEDER_1_UNIT_02."HMI_Offsets Alarms and Warnings".StirrerSpeedNominalLine1_Max_Alarm, STIRRER_SPEED_WARN_LOW_LIMIT => "DB21003_POWDER_FEEDER_HMI_INTERLOCK".POWDER_FEEDER_1_UNIT_02."HMI_Offsets Alarms and Warnings".StirrerSpeedNominalLine1_Min_Warning, STIRRER_SPEED_ALRM_LOW_LIMIT => "DB21003_POWDER_FEEDER_HMI_INTERLOCK".POWDER_FEEDER_1_UNIT_02."HMI_Offsets Alarms and Warnings".StirrerSpeedNominalLine1_Min_Alarm, TEMP_ALRM_UP_LIMIT => "DB21003_POWDER_FEEDER_HMI_INTERLOCK".POWDER_FEEDER_1_UNIT_02."HMI_Offsets Alarms and Warnings".HopperTempNominalLine1_Max_Alarm, HOPPER_TEMP_MANUAL => "DB21003_POWDER_FEEDER_HMI_INTERLOCK".POWDER_FEEDER_1_UNIT_02."HMI_Values Setpoints".HopperTempNominalLine1, STIRRER_SPEED_MANUAL => "DB21003_POWDER_FEEDER_HMI_INTERLOCK".POWDER_FEEDER_1_UNIT_02."HMI_Values Setpoints".StirrerSpeedNominalLine1, DISC_SPEED_MANUAL => "DB21003_POWDER_FEEDER_HMI_INTERLOCK".POWDER_FEEDER_1_UNIT_02."HMI_Values Setpoints".DiskSpeedNominalLine1, GAS_FLOW_RATE_MANUAL => "DB21003_POWDER_FEEDER_HMI_INTERLOCK".POWDER_FEEDER_1_UNIT_02."HMI_Values Setpoints".CarrierGasNominalLine1, HOPPER_ON_REQ =>, HOPPER_OFF_REQ =>, HEATER_ON_REQ =>, HEATER_OFF_REQ =>, START_SEQUENCE_GAS_STEPS => "DB21023_PF_1_HOPPERS_UNIT_02".SWITCH_ON_SEQUENCE_LINE_1.MAX_STEPS_GAS, START_SEQUENCE_DISK_STEPS => "DB21023_PF_1_HOPPERS_UNIT_02".SWITCH_ON_SEQUENCE_LINE_1.MAX_STEPS_DISK, STOP_SEQUENCE_GAS_STEPS => "DB21023_PF_1_HOPPERS_UNIT_02".SWITCH_OFF_SEQUENCE_LINE_1.MAX_STEPS_GAS, STOP_SEQUENCE_DISK_STEP => "DB21023_PF_1_HOPPERS_UNIT_02".SWITCH_OFF_SEQUENCE_LINE_1.MAX_STEPS_DISK, STOP_SEQUENCE_PAUSE_STEP => "DB21023_PF_1_HOPPERS_UNIT_02".SWITCH_OFF_SEQUENCE_LINE_1.GAS_WAIT_STEP, SELECTED_ARGON_GAS => "DB21003_POWDER_FEEDER_HMI_INTERLOCK".POWDER_FEEDER_1_UNIT_02.HMI_ACTIONS_STATUS.SELECTED_ARGON_GAS, SELECTED_NITROGEN_GAS => "DB21003_POWDER_FEEDER_HMI_INTERLOCK".POWDER_FEEDER_1_UNIT_02.HMI_ACTIONS_STATUS.SELECTED_NITROGEN_GAS, SELECTED_HELIUM_GAS => "DB21003_POWDER_FEEDER_HMI_INTERLOCK".POWDER_FEEDER_1_UNIT_02.HMI_ACTIONS_STATUS.SELECTED_HELIUM_GAS, SELECTED_ARGON30_GAS => "DB21003_POWDER_FEEDER_HMI_INTERLOCK".POWDER_FEEDER_1_UNIT_02.HMI_ACTIONS_STATUS.SELECTED_ARGON30_GAS)
   END_RUNG
   // the same network as SCL:
   "DB7250_FEEDER_1_UNIT_02_LINE_1"(GAS_FLOW_RATE_ACTUAL := "DB21005_POWDER_FEEDER_PLC_AUX"."INTERLOCKS_PLC_I/O_PF_1_UNIT_02".i_rCarriergasActual_Line1,   // "FB7238_VARIABLES_PLC_HMI_FEEDERS"
                           GAS_FLOW_RATE_AUTO := "DB7300_INTERLOCK".POWDER_FEEDERS.UNIT_02.POWDER_FEEDER_1_UNIT_02.CarrierGasNominalLine1,
                           DISC_SPEED_ACTUAL := "DB21005_POWDER_FEEDER_PLC_AUX"."INTERLOCKS_PLC_I/O_PF_1_UNIT_02".i_rDiskActual_Line1,
                           DISC_SPEED_AUTO := "DB7300_INTERLOCK".POWDER_FEEDERS.UNIT_02.POWDER_FEEDER_1_UNIT_02.DiskSpeedNominalLine1,
                           STIRRER_SPEED_ACTUAL := "DB21005_POWDER_FEEDER_PLC_AUX"."INTERLOCKS_PLC_I/O_PF_1_UNIT_02".i_rStirrerActual_Line1,
                           STIRRER_SPEED_AUTO := "DB7300_INTERLOCK".POWDER_FEEDERS.UNIT_02.POWDER_FEEDER_1_UNIT_02.StirrerSpeedNominalLine1,
                           HOPPER_TEMP_ACTUAL := "DB21005_POWDER_FEEDER_PLC_AUX"."INTERLOCKS_PLC_I/O_PF_1_UNIT_02".i_rHopperTempActual_Line1,
                           HOPPER_TEMP_AUTO := "DB7300_INTERLOCK".POWDER_FEEDERS.UNIT_02.POWDER_FEEDER_1_UNIT_02.HopperTempNominalLine1,
                           HEATER_STATUS := "DB21021_PF_1_HEATER_JKL_UNIT_02".HEATER_STATUS_LINE_1,
                           HOPPER_STATUS := "DB21023_PF_1_HOPPERS_UNIT_02".HOPPER_STATUS_LINE_1,
                           SELECTED_GAS := "DB7238_VARIABLES_PLC_CONNECTION".FEEDER_1_U02_SELECTED_GAS,
                           FEEDER_LINE_OUT := "DB7238_VARIABLES_PLC_CONNECTION".FEEDER_1_U_02_LINE_1,
                           HEATER_ON => "DB2040_WINCC_HMI_LINES".SERVICES[7].WINCC_LINE_REQUEST_RIGHT,
                           DISC_SPEED_WARN_UP_LIMIT => "DB21003_POWDER_FEEDER_HMI_INTERLOCK".POWDER_FEEDER_1_UNIT_02."HMI_Offsets Alarms and Warnings".DiskSpeedNominalLine1_Max_Warning,
                           DISC_SPEED_ALRM_UP_LIMIT => "DB21003_POWDER_FEEDER_HMI_INTERLOCK".POWDER_FEEDER_1_UNIT_02."HMI_Offsets Alarms and Warnings".DiskSpeedNominalLine1_Max_Alarm,
                           DISC_SPEED_WARN_LOW_LIMIT => "DB21003_POWDER_FEEDER_HMI_INTERLOCK".POWDER_FEEDER_1_UNIT_02."HMI_Offsets Alarms and Warnings".DiskSpeedNominalLine1_Min_Warning,
                           DISC_SPEED_ALRM_LOW_LIMIT => "DB21003_POWDER_FEEDER_HMI_INTERLOCK".POWDER_FEEDER_1_UNIT_02."HMI_Offsets Alarms and Warnings".DiskSpeedNominalLine1_Min_Alarm,
                           GAS_FLOW_RATE_WARN_UP_LIMIT => "DB21003_POWDER_FEEDER_HMI_INTERLOCK".POWDER_FEEDER_1_UNIT_02."HMI_Offsets Alarms and Warnings".CarrierGasNominalLine1_Max_Warning,
                           GAS_FLOW_RATE_ALRM_UP_LIMIT => "DB21003_POWDER_FEEDER_HMI_INTERLOCK".POWDER_FEEDER_1_UNIT_02."HMI_Offsets Alarms and Warnings".CarrierGasNominalLine1_Max_Alarm,
                           GAS_FLOW_RATE_WARN_LOW_LIMIT => "DB21003_POWDER_FEEDER_HMI_INTERLOCK".POWDER_FEEDER_1_UNIT_02."HMI_Offsets Alarms and Warnings".CarrierGasNominalLine1_Min_Warning,
                           GAS_FLOW_RATE_ALRM_LOW_LIMIT => "DB21003_POWDER_FEEDER_HMI_INTERLOCK".POWDER_FEEDER_1_UNIT_02."HMI_Offsets Alarms and Warnings".CarrierGasNominalLine1_Min_Alarm,
                           STIRRER_SPEED_WARN_UP_LIMIT => "DB21003_POWDER_FEEDER_HMI_INTERLOCK".POWDER_FEEDER_1_UNIT_02."HMI_Offsets Alarms and Warnings".StirrerSpeedNominalLine1_Max_Warning,
                           STIRRER_SPEED_ALRM_UP_LIMIT => "DB21003_POWDER_FEEDER_HMI_INTERLOCK".POWDER_FEEDER_1_UNIT_02."HMI_Offsets Alarms and Warnings".StirrerSpeedNominalLine1_Max_Alarm,
                           STIRRER_SPEED_WARN_LOW_LIMIT => "DB21003_POWDER_FEEDER_HMI_INTERLOCK".POWDER_FEEDER_1_UNIT_02."HMI_Offsets Alarms and Warnings".StirrerSpeedNominalLine1_Min_Warning,
                           STIRRER_SPEED_ALRM_LOW_LIMIT => "DB21003_POWDER_FEEDER_HMI_INTERLOCK".POWDER_FEEDER_1_UNIT_02."HMI_Offsets Alarms and Warnings".StirrerSpeedNominalLine1_Min_Alarm,
                           TEMP_ALRM_UP_LIMIT => "DB21003_POWDER_FEEDER_HMI_INTERLOCK".POWDER_FEEDER_1_UNIT_02."HMI_Offsets Alarms and Warnings".HopperTempNominalLine1_Max_Alarm,
                           HOPPER_TEMP_MANUAL => "DB21003_POWDER_FEEDER_HMI_INTERLOCK".POWDER_FEEDER_1_UNIT_02."HMI_Values Setpoints".HopperTempNominalLine1,
                           STIRRER_SPEED_MANUAL => "DB21003_POWDER_FEEDER_HMI_INTERLOCK".POWDER_FEEDER_1_UNIT_02."HMI_Values Setpoints".StirrerSpeedNominalLine1,
                           DISC_SPEED_MANUAL => "DB21003_POWDER_FEEDER_HMI_INTERLOCK".POWDER_FEEDER_1_UNIT_02."HMI_Values Setpoints".DiskSpeedNominalLine1,
                           GAS_FLOW_RATE_MANUAL => "DB21003_POWDER_FEEDER_HMI_INTERLOCK".POWDER_FEEDER_1_UNIT_02."HMI_Values Setpoints".CarrierGasNominalLine1,
                           START_SEQUENCE_GAS_STEPS => "DB21023_PF_1_HOPPERS_UNIT_02".SWITCH_ON_SEQUENCE_LINE_1.MAX_STEPS_GAS,
                           START_SEQUENCE_DISK_STEPS => "DB21023_PF_1_HOPPERS_UNIT_02".SWITCH_ON_SEQUENCE_LINE_1.MAX_STEPS_DISK,
                           STOP_SEQUENCE_GAS_STEPS => "DB21023_PF_1_HOPPERS_UNIT_02".SWITCH_OFF_SEQUENCE_LINE_1.MAX_STEPS_GAS,
                           STOP_SEQUENCE_DISK_STEP => "DB21023_PF_1_HOPPERS_UNIT_02".SWITCH_OFF_SEQUENCE_LINE_1.MAX_STEPS_DISK,
                           STOP_SEQUENCE_PAUSE_STEP => "DB21023_PF_1_HOPPERS_UNIT_02".SWITCH_OFF_SEQUENCE_LINE_1.GAS_WAIT_STEP,
                           SELECTED_ARGON_GAS => "DB21003_POWDER_FEEDER_HMI_INTERLOCK".POWDER_FEEDER_1_UNIT_02.HMI_ACTIONS_STATUS.SELECTED_ARGON_GAS,
                           SELECTED_NITROGEN_GAS => "DB21003_POWDER_FEEDER_HMI_INTERLOCK".POWDER_FEEDER_1_UNIT_02.HMI_ACTIONS_STATUS.SELECTED_NITROGEN_GAS,
                           SELECTED_HELIUM_GAS => "DB21003_POWDER_FEEDER_HMI_INTERLOCK".POWDER_FEEDER_1_UNIT_02.HMI_ACTIONS_STATUS.SELECTED_HELIUM_GAS,
                           SELECTED_ARGON30_GAS => "DB21003_POWDER_FEEDER_HMI_INTERLOCK".POWDER_FEEDER_1_UNIT_02.HMI_ACTIONS_STATUS.SELECTED_ARGON30_GAS);
END_REGION

REGION Network 5: FEEDER 1 UNIT 02 LINE 2
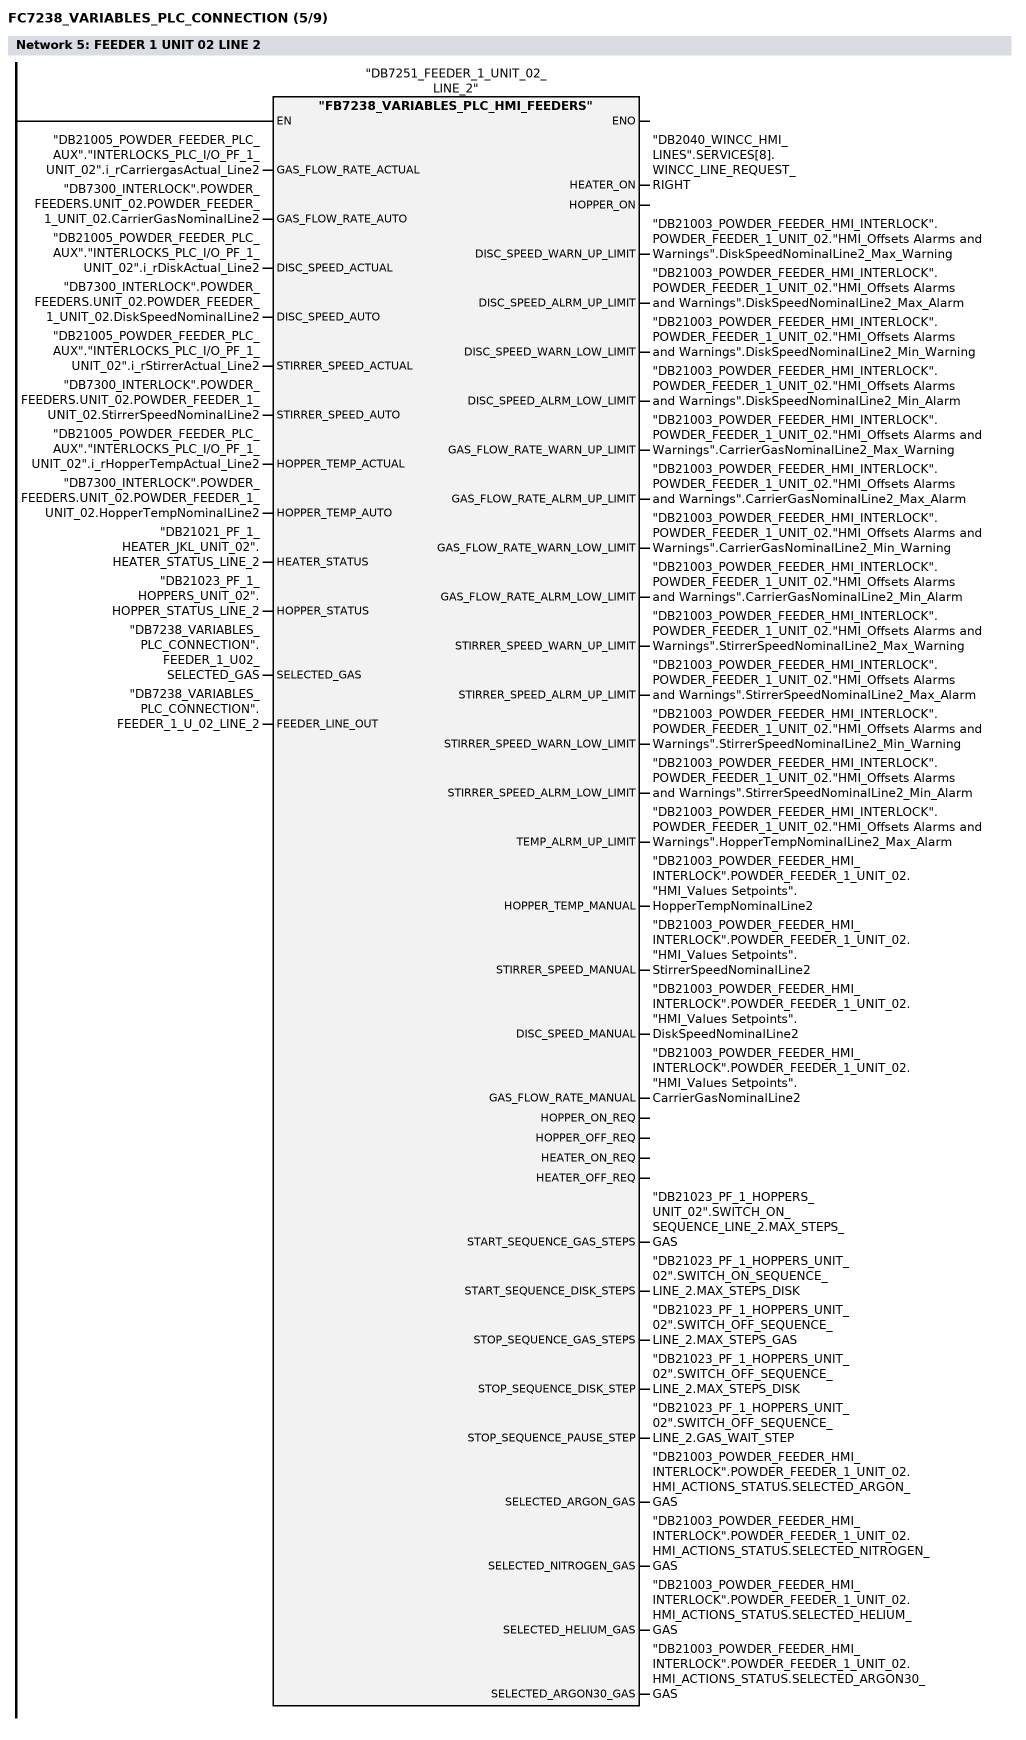
   RUNG wire#powerrail
      "DB7251_FEEDER_1_UNIT_02_LINE_2"(GAS_FLOW_RATE_ACTUAL := "DB21005_POWDER_FEEDER_PLC_AUX"."INTERLOCKS_PLC_I/O_PF_1_UNIT_02".i_rCarriergasActual_Line2, GAS_FLOW_RATE_AUTO := "DB7300_INTERLOCK".POWDER_FEEDERS.UNIT_02.POWDER_FEEDER_1_UNIT_02.CarrierGasNominalLine2, DISC_SPEED_ACTUAL := "DB21005_POWDER_FEEDER_PLC_AUX"."INTERLOCKS_PLC_I/O_PF_1_UNIT_02".i_rDiskActual_Line2, DISC_SPEED_AUTO := "DB7300_INTERLOCK".POWDER_FEEDERS.UNIT_02.POWDER_FEEDER_1_UNIT_02.DiskSpeedNominalLine2, STIRRER_SPEED_ACTUAL := "DB21005_POWDER_FEEDER_PLC_AUX"."INTERLOCKS_PLC_I/O_PF_1_UNIT_02".i_rStirrerActual_Line2, STIRRER_SPEED_AUTO := "DB7300_INTERLOCK".POWDER_FEEDERS.UNIT_02.POWDER_FEEDER_1_UNIT_02.StirrerSpeedNominalLine2, HOPPER_TEMP_ACTUAL := "DB21005_POWDER_FEEDER_PLC_AUX"."INTERLOCKS_PLC_I/O_PF_1_UNIT_02".i_rHopperTempActual_Line2, HOPPER_TEMP_AUTO := "DB7300_INTERLOCK".POWDER_FEEDERS.UNIT_02.POWDER_FEEDER_1_UNIT_02.HopperTempNominalLine2, HEATER_STATUS := "DB21021_PF_1_HEATER_JKL_UNIT_02".HEATER_STATUS_LINE_2, HOPPER_STATUS := "DB21023_PF_1_HOPPERS_UNIT_02".HOPPER_STATUS_LINE_2, SELECTED_GAS := "DB7238_VARIABLES_PLC_CONNECTION".FEEDER_1_U02_SELECTED_GAS, FEEDER_LINE_OUT := "DB7238_VARIABLES_PLC_CONNECTION".FEEDER_1_U_02_LINE_2, HEATER_ON => "DB2040_WINCC_HMI_LINES".SERVICES[8].WINCC_LINE_REQUEST_RIGHT, HOPPER_ON =>, DISC_SPEED_WARN_UP_LIMIT => "DB21003_POWDER_FEEDER_HMI_INTERLOCK".POWDER_FEEDER_1_UNIT_02."HMI_Offsets Alarms and Warnings".DiskSpeedNominalLine2_Max_Warning, DISC_SPEED_ALRM_UP_LIMIT => "DB21003_POWDER_FEEDER_HMI_INTERLOCK".POWDER_FEEDER_1_UNIT_02."HMI_Offsets Alarms and Warnings".DiskSpeedNominalLine2_Max_Alarm, DISC_SPEED_WARN_LOW_LIMIT => "DB21003_POWDER_FEEDER_HMI_INTERLOCK".POWDER_FEEDER_1_UNIT_02."HMI_Offsets Alarms and Warnings".DiskSpeedNominalLine2_Min_Warning, DISC_SPEED_ALRM_LOW_LIMIT => "DB21003_POWDER_FEEDER_HMI_INTERLOCK".POWDER_FEEDER_1_UNIT_02."HMI_Offsets Alarms and Warnings".DiskSpeedNominalLine2_Min_Alarm, GAS_FLOW_RATE_WARN_UP_LIMIT => "DB21003_POWDER_FEEDER_HMI_INTERLOCK".POWDER_FEEDER_1_UNIT_02."HMI_Offsets Alarms and Warnings".CarrierGasNominalLine2_Max_Warning, GAS_FLOW_RATE_ALRM_UP_LIMIT => "DB21003_POWDER_FEEDER_HMI_INTERLOCK".POWDER_FEEDER_1_UNIT_02."HMI_Offsets Alarms and Warnings".CarrierGasNominalLine2_Max_Alarm, GAS_FLOW_RATE_WARN_LOW_LIMIT => "DB21003_POWDER_FEEDER_HMI_INTERLOCK".POWDER_FEEDER_1_UNIT_02."HMI_Offsets Alarms and Warnings".CarrierGasNominalLine2_Min_Warning, GAS_FLOW_RATE_ALRM_LOW_LIMIT => "DB21003_POWDER_FEEDER_HMI_INTERLOCK".POWDER_FEEDER_1_UNIT_02."HMI_Offsets Alarms and Warnings".CarrierGasNominalLine2_Min_Alarm, STIRRER_SPEED_WARN_UP_LIMIT => "DB21003_POWDER_FEEDER_HMI_INTERLOCK".POWDER_FEEDER_1_UNIT_02."HMI_Offsets Alarms and Warnings".StirrerSpeedNominalLine2_Max_Warning, STIRRER_SPEED_ALRM_UP_LIMIT => "DB21003_POWDER_FEEDER_HMI_INTERLOCK".POWDER_FEEDER_1_UNIT_02."HMI_Offsets Alarms and Warnings".StirrerSpeedNominalLine2_Max_Alarm, STIRRER_SPEED_WARN_LOW_LIMIT => "DB21003_POWDER_FEEDER_HMI_INTERLOCK".POWDER_FEEDER_1_UNIT_02."HMI_Offsets Alarms and Warnings".StirrerSpeedNominalLine2_Min_Warning, STIRRER_SPEED_ALRM_LOW_LIMIT => "DB21003_POWDER_FEEDER_HMI_INTERLOCK".POWDER_FEEDER_1_UNIT_02."HMI_Offsets Alarms and Warnings".StirrerSpeedNominalLine2_Min_Alarm, TEMP_ALRM_UP_LIMIT => "DB21003_POWDER_FEEDER_HMI_INTERLOCK".POWDER_FEEDER_1_UNIT_02."HMI_Offsets Alarms and Warnings".HopperTempNominalLine2_Max_Alarm, HOPPER_TEMP_MANUAL => "DB21003_POWDER_FEEDER_HMI_INTERLOCK".POWDER_FEEDER_1_UNIT_02."HMI_Values Setpoints".HopperTempNominalLine2, STIRRER_SPEED_MANUAL => "DB21003_POWDER_FEEDER_HMI_INTERLOCK".POWDER_FEEDER_1_UNIT_02."HMI_Values Setpoints".StirrerSpeedNominalLine2, DISC_SPEED_MANUAL => "DB21003_POWDER_FEEDER_HMI_INTERLOCK".POWDER_FEEDER_1_UNIT_02."HMI_Values Setpoints".DiskSpeedNominalLine2, GAS_FLOW_RATE_MANUAL => "DB21003_POWDER_FEEDER_HMI_INTERLOCK".POWDER_FEEDER_1_UNIT_02."HMI_Values Setpoints".CarrierGasNominalLine2, HOPPER_ON_REQ =>, HOPPER_OFF_REQ =>, HEATER_ON_REQ =>, HEATER_OFF_REQ =>, START_SEQUENCE_GAS_STEPS => "DB21023_PF_1_HOPPERS_UNIT_02".SWITCH_ON_SEQUENCE_LINE_2.MAX_STEPS_GAS, START_SEQUENCE_DISK_STEPS => "DB21023_PF_1_HOPPERS_UNIT_02".SWITCH_ON_SEQUENCE_LINE_2.MAX_STEPS_DISK, STOP_SEQUENCE_GAS_STEPS => "DB21023_PF_1_HOPPERS_UNIT_02".SWITCH_OFF_SEQUENCE_LINE_2.MAX_STEPS_GAS, STOP_SEQUENCE_DISK_STEP => "DB21023_PF_1_HOPPERS_UNIT_02".SWITCH_OFF_SEQUENCE_LINE_2.MAX_STEPS_DISK, STOP_SEQUENCE_PAUSE_STEP => "DB21023_PF_1_HOPPERS_UNIT_02".SWITCH_OFF_SEQUENCE_LINE_2.GAS_WAIT_STEP, SELECTED_ARGON_GAS => "DB21003_POWDER_FEEDER_HMI_INTERLOCK".POWDER_FEEDER_1_UNIT_02.HMI_ACTIONS_STATUS.SELECTED_ARGON_GAS, SELECTED_NITROGEN_GAS => "DB21003_POWDER_FEEDER_HMI_INTERLOCK".POWDER_FEEDER_1_UNIT_02.HMI_ACTIONS_STATUS.SELECTED_NITROGEN_GAS, SELECTED_HELIUM_GAS => "DB21003_POWDER_FEEDER_HMI_INTERLOCK".POWDER_FEEDER_1_UNIT_02.HMI_ACTIONS_STATUS.SELECTED_HELIUM_GAS, SELECTED_ARGON30_GAS => "DB21003_POWDER_FEEDER_HMI_INTERLOCK".POWDER_FEEDER_1_UNIT_02.HMI_ACTIONS_STATUS.SELECTED_ARGON30_GAS)
   END_RUNG
   // the same network as SCL:
   "DB7251_FEEDER_1_UNIT_02_LINE_2"(GAS_FLOW_RATE_ACTUAL := "DB21005_POWDER_FEEDER_PLC_AUX"."INTERLOCKS_PLC_I/O_PF_1_UNIT_02".i_rCarriergasActual_Line2,   // "FB7238_VARIABLES_PLC_HMI_FEEDERS"
                           GAS_FLOW_RATE_AUTO := "DB7300_INTERLOCK".POWDER_FEEDERS.UNIT_02.POWDER_FEEDER_1_UNIT_02.CarrierGasNominalLine2,
                           DISC_SPEED_ACTUAL := "DB21005_POWDER_FEEDER_PLC_AUX"."INTERLOCKS_PLC_I/O_PF_1_UNIT_02".i_rDiskActual_Line2,
                           DISC_SPEED_AUTO := "DB7300_INTERLOCK".POWDER_FEEDERS.UNIT_02.POWDER_FEEDER_1_UNIT_02.DiskSpeedNominalLine2,
                           STIRRER_SPEED_ACTUAL := "DB21005_POWDER_FEEDER_PLC_AUX"."INTERLOCKS_PLC_I/O_PF_1_UNIT_02".i_rStirrerActual_Line2,
                           STIRRER_SPEED_AUTO := "DB7300_INTERLOCK".POWDER_FEEDERS.UNIT_02.POWDER_FEEDER_1_UNIT_02.StirrerSpeedNominalLine2,
                           HOPPER_TEMP_ACTUAL := "DB21005_POWDER_FEEDER_PLC_AUX"."INTERLOCKS_PLC_I/O_PF_1_UNIT_02".i_rHopperTempActual_Line2,
                           HOPPER_TEMP_AUTO := "DB7300_INTERLOCK".POWDER_FEEDERS.UNIT_02.POWDER_FEEDER_1_UNIT_02.HopperTempNominalLine2,
                           HEATER_STATUS := "DB21021_PF_1_HEATER_JKL_UNIT_02".HEATER_STATUS_LINE_2,
                           HOPPER_STATUS := "DB21023_PF_1_HOPPERS_UNIT_02".HOPPER_STATUS_LINE_2,
                           SELECTED_GAS := "DB7238_VARIABLES_PLC_CONNECTION".FEEDER_1_U02_SELECTED_GAS,
                           FEEDER_LINE_OUT := "DB7238_VARIABLES_PLC_CONNECTION".FEEDER_1_U_02_LINE_2,
                           HEATER_ON => "DB2040_WINCC_HMI_LINES".SERVICES[8].WINCC_LINE_REQUEST_RIGHT,
                           DISC_SPEED_WARN_UP_LIMIT => "DB21003_POWDER_FEEDER_HMI_INTERLOCK".POWDER_FEEDER_1_UNIT_02."HMI_Offsets Alarms and Warnings".DiskSpeedNominalLine2_Max_Warning,
                           DISC_SPEED_ALRM_UP_LIMIT => "DB21003_POWDER_FEEDER_HMI_INTERLOCK".POWDER_FEEDER_1_UNIT_02."HMI_Offsets Alarms and Warnings".DiskSpeedNominalLine2_Max_Alarm,
                           DISC_SPEED_WARN_LOW_LIMIT => "DB21003_POWDER_FEEDER_HMI_INTERLOCK".POWDER_FEEDER_1_UNIT_02."HMI_Offsets Alarms and Warnings".DiskSpeedNominalLine2_Min_Warning,
                           DISC_SPEED_ALRM_LOW_LIMIT => "DB21003_POWDER_FEEDER_HMI_INTERLOCK".POWDER_FEEDER_1_UNIT_02."HMI_Offsets Alarms and Warnings".DiskSpeedNominalLine2_Min_Alarm,
                           GAS_FLOW_RATE_WARN_UP_LIMIT => "DB21003_POWDER_FEEDER_HMI_INTERLOCK".POWDER_FEEDER_1_UNIT_02."HMI_Offsets Alarms and Warnings".CarrierGasNominalLine2_Max_Warning,
                           GAS_FLOW_RATE_ALRM_UP_LIMIT => "DB21003_POWDER_FEEDER_HMI_INTERLOCK".POWDER_FEEDER_1_UNIT_02."HMI_Offsets Alarms and Warnings".CarrierGasNominalLine2_Max_Alarm,
                           GAS_FLOW_RATE_WARN_LOW_LIMIT => "DB21003_POWDER_FEEDER_HMI_INTERLOCK".POWDER_FEEDER_1_UNIT_02."HMI_Offsets Alarms and Warnings".CarrierGasNominalLine2_Min_Warning,
                           GAS_FLOW_RATE_ALRM_LOW_LIMIT => "DB21003_POWDER_FEEDER_HMI_INTERLOCK".POWDER_FEEDER_1_UNIT_02."HMI_Offsets Alarms and Warnings".CarrierGasNominalLine2_Min_Alarm,
                           STIRRER_SPEED_WARN_UP_LIMIT => "DB21003_POWDER_FEEDER_HMI_INTERLOCK".POWDER_FEEDER_1_UNIT_02."HMI_Offsets Alarms and Warnings".StirrerSpeedNominalLine2_Max_Warning,
                           STIRRER_SPEED_ALRM_UP_LIMIT => "DB21003_POWDER_FEEDER_HMI_INTERLOCK".POWDER_FEEDER_1_UNIT_02."HMI_Offsets Alarms and Warnings".StirrerSpeedNominalLine2_Max_Alarm,
                           STIRRER_SPEED_WARN_LOW_LIMIT => "DB21003_POWDER_FEEDER_HMI_INTERLOCK".POWDER_FEEDER_1_UNIT_02."HMI_Offsets Alarms and Warnings".StirrerSpeedNominalLine2_Min_Warning,
                           STIRRER_SPEED_ALRM_LOW_LIMIT => "DB21003_POWDER_FEEDER_HMI_INTERLOCK".POWDER_FEEDER_1_UNIT_02."HMI_Offsets Alarms and Warnings".StirrerSpeedNominalLine2_Min_Alarm,
                           TEMP_ALRM_UP_LIMIT => "DB21003_POWDER_FEEDER_HMI_INTERLOCK".POWDER_FEEDER_1_UNIT_02."HMI_Offsets Alarms and Warnings".HopperTempNominalLine2_Max_Alarm,
                           HOPPER_TEMP_MANUAL => "DB21003_POWDER_FEEDER_HMI_INTERLOCK".POWDER_FEEDER_1_UNIT_02."HMI_Values Setpoints".HopperTempNominalLine2,
                           STIRRER_SPEED_MANUAL => "DB21003_POWDER_FEEDER_HMI_INTERLOCK".POWDER_FEEDER_1_UNIT_02."HMI_Values Setpoints".StirrerSpeedNominalLine2,
                           DISC_SPEED_MANUAL => "DB21003_POWDER_FEEDER_HMI_INTERLOCK".POWDER_FEEDER_1_UNIT_02."HMI_Values Setpoints".DiskSpeedNominalLine2,
                           GAS_FLOW_RATE_MANUAL => "DB21003_POWDER_FEEDER_HMI_INTERLOCK".POWDER_FEEDER_1_UNIT_02."HMI_Values Setpoints".CarrierGasNominalLine2,
                           START_SEQUENCE_GAS_STEPS => "DB21023_PF_1_HOPPERS_UNIT_02".SWITCH_ON_SEQUENCE_LINE_2.MAX_STEPS_GAS,
                           START_SEQUENCE_DISK_STEPS => "DB21023_PF_1_HOPPERS_UNIT_02".SWITCH_ON_SEQUENCE_LINE_2.MAX_STEPS_DISK,
                           STOP_SEQUENCE_GAS_STEPS => "DB21023_PF_1_HOPPERS_UNIT_02".SWITCH_OFF_SEQUENCE_LINE_2.MAX_STEPS_GAS,
                           STOP_SEQUENCE_DISK_STEP => "DB21023_PF_1_HOPPERS_UNIT_02".SWITCH_OFF_SEQUENCE_LINE_2.MAX_STEPS_DISK,
                           STOP_SEQUENCE_PAUSE_STEP => "DB21023_PF_1_HOPPERS_UNIT_02".SWITCH_OFF_SEQUENCE_LINE_2.GAS_WAIT_STEP,
                           SELECTED_ARGON_GAS => "DB21003_POWDER_FEEDER_HMI_INTERLOCK".POWDER_FEEDER_1_UNIT_02.HMI_ACTIONS_STATUS.SELECTED_ARGON_GAS,
                           SELECTED_NITROGEN_GAS => "DB21003_POWDER_FEEDER_HMI_INTERLOCK".POWDER_FEEDER_1_UNIT_02.HMI_ACTIONS_STATUS.SELECTED_NITROGEN_GAS,
                           SELECTED_HELIUM_GAS => "DB21003_POWDER_FEEDER_HMI_INTERLOCK".POWDER_FEEDER_1_UNIT_02.HMI_ACTIONS_STATUS.SELECTED_HELIUM_GAS,
                           SELECTED_ARGON30_GAS => "DB21003_POWDER_FEEDER_HMI_INTERLOCK".POWDER_FEEDER_1_UNIT_02.HMI_ACTIONS_STATUS.SELECTED_ARGON30_GAS);
END_REGION

REGION Network 6: FEEDER 2 UNIT 02 LINE 2
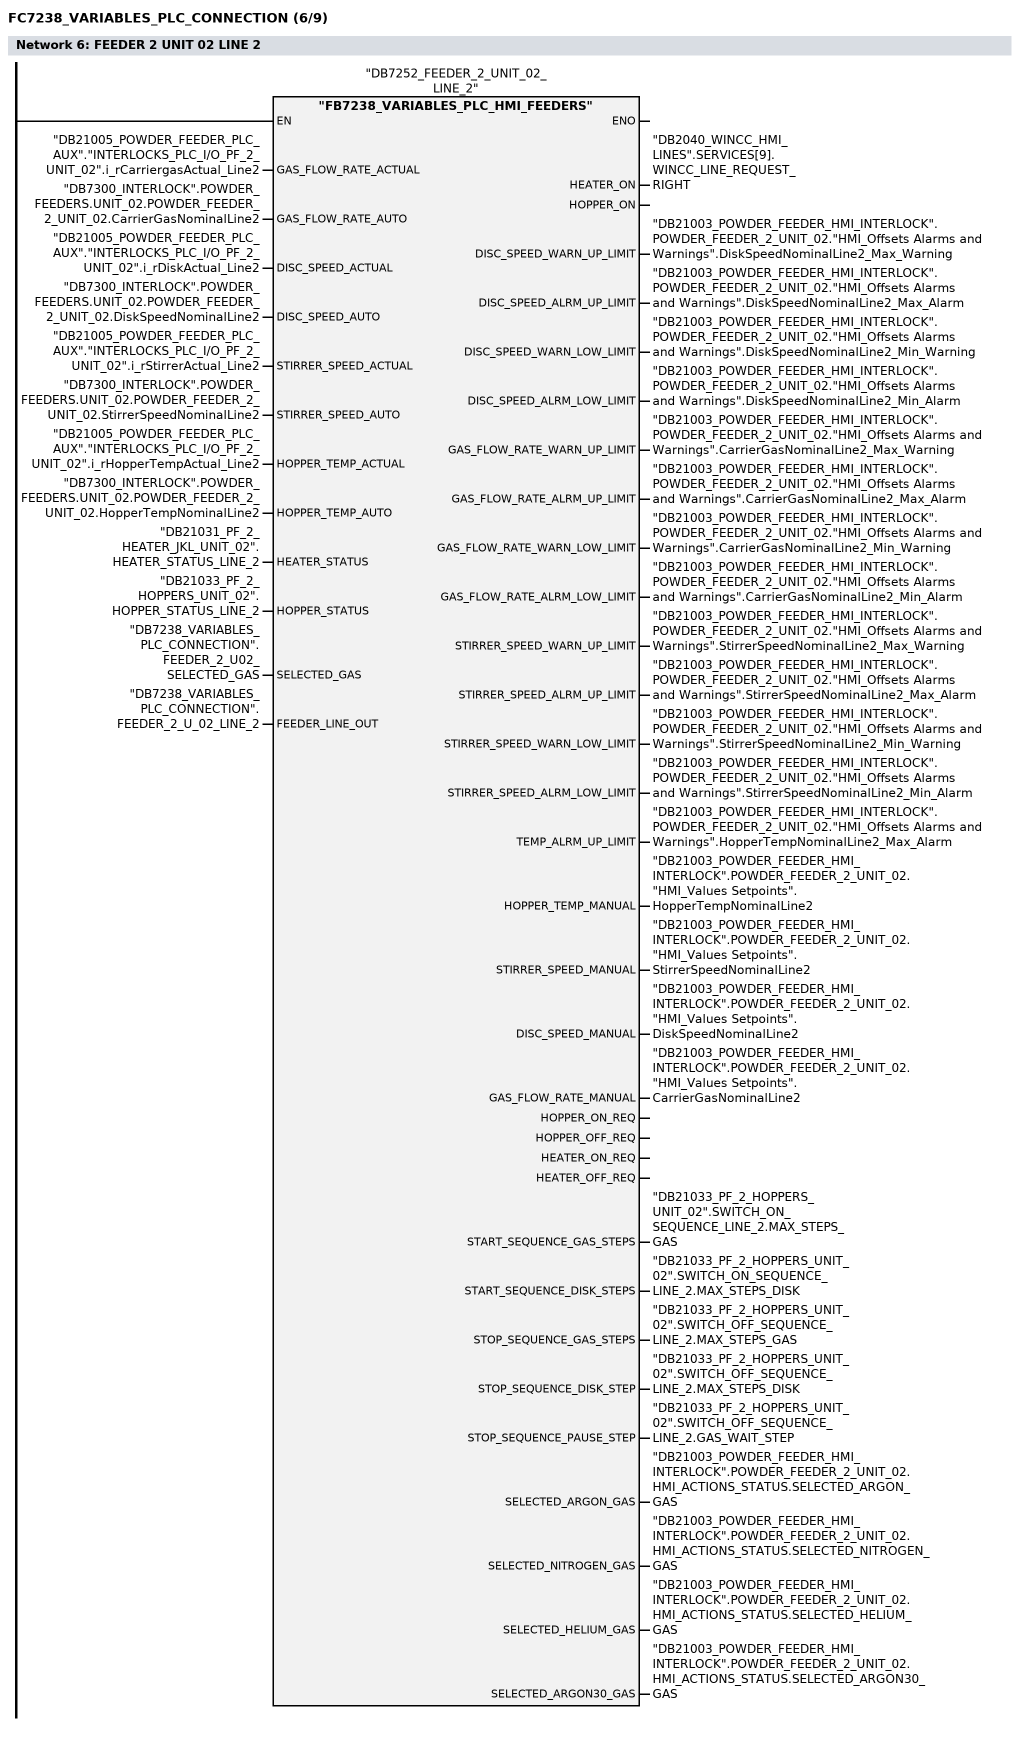
   RUNG wire#powerrail
      "DB7252_FEEDER_2_UNIT_02_LINE_2"(GAS_FLOW_RATE_ACTUAL := "DB21005_POWDER_FEEDER_PLC_AUX"."INTERLOCKS_PLC_I/O_PF_2_UNIT_02".i_rCarriergasActual_Line2, GAS_FLOW_RATE_AUTO := "DB7300_INTERLOCK".POWDER_FEEDERS.UNIT_02.POWDER_FEEDER_2_UNIT_02.CarrierGasNominalLine2, DISC_SPEED_ACTUAL := "DB21005_POWDER_FEEDER_PLC_AUX"."INTERLOCKS_PLC_I/O_PF_2_UNIT_02".i_rDiskActual_Line2, DISC_SPEED_AUTO := "DB7300_INTERLOCK".POWDER_FEEDERS.UNIT_02.POWDER_FEEDER_2_UNIT_02.DiskSpeedNominalLine2, STIRRER_SPEED_ACTUAL := "DB21005_POWDER_FEEDER_PLC_AUX"."INTERLOCKS_PLC_I/O_PF_2_UNIT_02".i_rStirrerActual_Line2, STIRRER_SPEED_AUTO := "DB7300_INTERLOCK".POWDER_FEEDERS.UNIT_02.POWDER_FEEDER_2_UNIT_02.StirrerSpeedNominalLine2, HOPPER_TEMP_ACTUAL := "DB21005_POWDER_FEEDER_PLC_AUX"."INTERLOCKS_PLC_I/O_PF_2_UNIT_02".i_rHopperTempActual_Line2, HOPPER_TEMP_AUTO := "DB7300_INTERLOCK".POWDER_FEEDERS.UNIT_02.POWDER_FEEDER_2_UNIT_02.HopperTempNominalLine2, HEATER_STATUS := "DB21031_PF_2_HEATER_JKL_UNIT_02".HEATER_STATUS_LINE_2, HOPPER_STATUS := "DB21033_PF_2_HOPPERS_UNIT_02".HOPPER_STATUS_LINE_2, SELECTED_GAS := "DB7238_VARIABLES_PLC_CONNECTION".FEEDER_2_U02_SELECTED_GAS, FEEDER_LINE_OUT := "DB7238_VARIABLES_PLC_CONNECTION".FEEDER_2_U_02_LINE_2, HEATER_ON => "DB2040_WINCC_HMI_LINES".SERVICES[9].WINCC_LINE_REQUEST_RIGHT, HOPPER_ON =>, DISC_SPEED_WARN_UP_LIMIT => "DB21003_POWDER_FEEDER_HMI_INTERLOCK".POWDER_FEEDER_2_UNIT_02."HMI_Offsets Alarms and Warnings".DiskSpeedNominalLine2_Max_Warning, DISC_SPEED_ALRM_UP_LIMIT => "DB21003_POWDER_FEEDER_HMI_INTERLOCK".POWDER_FEEDER_2_UNIT_02."HMI_Offsets Alarms and Warnings".DiskSpeedNominalLine2_Max_Alarm, DISC_SPEED_WARN_LOW_LIMIT => "DB21003_POWDER_FEEDER_HMI_INTERLOCK".POWDER_FEEDER_2_UNIT_02."HMI_Offsets Alarms and Warnings".DiskSpeedNominalLine2_Min_Warning, DISC_SPEED_ALRM_LOW_LIMIT => "DB21003_POWDER_FEEDER_HMI_INTERLOCK".POWDER_FEEDER_2_UNIT_02."HMI_Offsets Alarms and Warnings".DiskSpeedNominalLine2_Min_Alarm, GAS_FLOW_RATE_WARN_UP_LIMIT => "DB21003_POWDER_FEEDER_HMI_INTERLOCK".POWDER_FEEDER_2_UNIT_02."HMI_Offsets Alarms and Warnings".CarrierGasNominalLine2_Max_Warning, GAS_FLOW_RATE_ALRM_UP_LIMIT => "DB21003_POWDER_FEEDER_HMI_INTERLOCK".POWDER_FEEDER_2_UNIT_02."HMI_Offsets Alarms and Warnings".CarrierGasNominalLine2_Max_Alarm, GAS_FLOW_RATE_WARN_LOW_LIMIT => "DB21003_POWDER_FEEDER_HMI_INTERLOCK".POWDER_FEEDER_2_UNIT_02."HMI_Offsets Alarms and Warnings".CarrierGasNominalLine2_Min_Warning, GAS_FLOW_RATE_ALRM_LOW_LIMIT => "DB21003_POWDER_FEEDER_HMI_INTERLOCK".POWDER_FEEDER_2_UNIT_02."HMI_Offsets Alarms and Warnings".CarrierGasNominalLine2_Min_Alarm, STIRRER_SPEED_WARN_UP_LIMIT => "DB21003_POWDER_FEEDER_HMI_INTERLOCK".POWDER_FEEDER_2_UNIT_02."HMI_Offsets Alarms and Warnings".StirrerSpeedNominalLine2_Max_Warning, STIRRER_SPEED_ALRM_UP_LIMIT => "DB21003_POWDER_FEEDER_HMI_INTERLOCK".POWDER_FEEDER_2_UNIT_02."HMI_Offsets Alarms and Warnings".StirrerSpeedNominalLine2_Max_Alarm, STIRRER_SPEED_WARN_LOW_LIMIT => "DB21003_POWDER_FEEDER_HMI_INTERLOCK".POWDER_FEEDER_2_UNIT_02."HMI_Offsets Alarms and Warnings".StirrerSpeedNominalLine2_Min_Warning, STIRRER_SPEED_ALRM_LOW_LIMIT => "DB21003_POWDER_FEEDER_HMI_INTERLOCK".POWDER_FEEDER_2_UNIT_02."HMI_Offsets Alarms and Warnings".StirrerSpeedNominalLine2_Min_Alarm, TEMP_ALRM_UP_LIMIT => "DB21003_POWDER_FEEDER_HMI_INTERLOCK".POWDER_FEEDER_2_UNIT_02."HMI_Offsets Alarms and Warnings".HopperTempNominalLine2_Max_Alarm, HOPPER_TEMP_MANUAL => "DB21003_POWDER_FEEDER_HMI_INTERLOCK".POWDER_FEEDER_2_UNIT_02."HMI_Values Setpoints".HopperTempNominalLine2, STIRRER_SPEED_MANUAL => "DB21003_POWDER_FEEDER_HMI_INTERLOCK".POWDER_FEEDER_2_UNIT_02."HMI_Values Setpoints".StirrerSpeedNominalLine2, DISC_SPEED_MANUAL => "DB21003_POWDER_FEEDER_HMI_INTERLOCK".POWDER_FEEDER_2_UNIT_02."HMI_Values Setpoints".DiskSpeedNominalLine2, GAS_FLOW_RATE_MANUAL => "DB21003_POWDER_FEEDER_HMI_INTERLOCK".POWDER_FEEDER_2_UNIT_02."HMI_Values Setpoints".CarrierGasNominalLine2, HOPPER_ON_REQ =>, HOPPER_OFF_REQ =>, HEATER_ON_REQ =>, HEATER_OFF_REQ =>, START_SEQUENCE_GAS_STEPS => "DB21033_PF_2_HOPPERS_UNIT_02".SWITCH_ON_SEQUENCE_LINE_2.MAX_STEPS_GAS, START_SEQUENCE_DISK_STEPS => "DB21033_PF_2_HOPPERS_UNIT_02".SWITCH_ON_SEQUENCE_LINE_2.MAX_STEPS_DISK, STOP_SEQUENCE_GAS_STEPS => "DB21033_PF_2_HOPPERS_UNIT_02".SWITCH_OFF_SEQUENCE_LINE_2.MAX_STEPS_GAS, STOP_SEQUENCE_DISK_STEP => "DB21033_PF_2_HOPPERS_UNIT_02".SWITCH_OFF_SEQUENCE_LINE_2.MAX_STEPS_DISK, STOP_SEQUENCE_PAUSE_STEP => "DB21033_PF_2_HOPPERS_UNIT_02".SWITCH_OFF_SEQUENCE_LINE_2.GAS_WAIT_STEP, SELECTED_ARGON_GAS => "DB21003_POWDER_FEEDER_HMI_INTERLOCK".POWDER_FEEDER_2_UNIT_02.HMI_ACTIONS_STATUS.SELECTED_ARGON_GAS, SELECTED_NITROGEN_GAS => "DB21003_POWDER_FEEDER_HMI_INTERLOCK".POWDER_FEEDER_2_UNIT_02.HMI_ACTIONS_STATUS.SELECTED_NITROGEN_GAS, SELECTED_HELIUM_GAS => "DB21003_POWDER_FEEDER_HMI_INTERLOCK".POWDER_FEEDER_2_UNIT_02.HMI_ACTIONS_STATUS.SELECTED_HELIUM_GAS, SELECTED_ARGON30_GAS => "DB21003_POWDER_FEEDER_HMI_INTERLOCK".POWDER_FEEDER_2_UNIT_02.HMI_ACTIONS_STATUS.SELECTED_ARGON30_GAS)
   END_RUNG
   // the same network as SCL:
   "DB7252_FEEDER_2_UNIT_02_LINE_2"(GAS_FLOW_RATE_ACTUAL := "DB21005_POWDER_FEEDER_PLC_AUX"."INTERLOCKS_PLC_I/O_PF_2_UNIT_02".i_rCarriergasActual_Line2,   // "FB7238_VARIABLES_PLC_HMI_FEEDERS"
                           GAS_FLOW_RATE_AUTO := "DB7300_INTERLOCK".POWDER_FEEDERS.UNIT_02.POWDER_FEEDER_2_UNIT_02.CarrierGasNominalLine2,
                           DISC_SPEED_ACTUAL := "DB21005_POWDER_FEEDER_PLC_AUX"."INTERLOCKS_PLC_I/O_PF_2_UNIT_02".i_rDiskActual_Line2,
                           DISC_SPEED_AUTO := "DB7300_INTERLOCK".POWDER_FEEDERS.UNIT_02.POWDER_FEEDER_2_UNIT_02.DiskSpeedNominalLine2,
                           STIRRER_SPEED_ACTUAL := "DB21005_POWDER_FEEDER_PLC_AUX"."INTERLOCKS_PLC_I/O_PF_2_UNIT_02".i_rStirrerActual_Line2,
                           STIRRER_SPEED_AUTO := "DB7300_INTERLOCK".POWDER_FEEDERS.UNIT_02.POWDER_FEEDER_2_UNIT_02.StirrerSpeedNominalLine2,
                           HOPPER_TEMP_ACTUAL := "DB21005_POWDER_FEEDER_PLC_AUX"."INTERLOCKS_PLC_I/O_PF_2_UNIT_02".i_rHopperTempActual_Line2,
                           HOPPER_TEMP_AUTO := "DB7300_INTERLOCK".POWDER_FEEDERS.UNIT_02.POWDER_FEEDER_2_UNIT_02.HopperTempNominalLine2,
                           HEATER_STATUS := "DB21031_PF_2_HEATER_JKL_UNIT_02".HEATER_STATUS_LINE_2,
                           HOPPER_STATUS := "DB21033_PF_2_HOPPERS_UNIT_02".HOPPER_STATUS_LINE_2,
                           SELECTED_GAS := "DB7238_VARIABLES_PLC_CONNECTION".FEEDER_2_U02_SELECTED_GAS,
                           FEEDER_LINE_OUT := "DB7238_VARIABLES_PLC_CONNECTION".FEEDER_2_U_02_LINE_2,
                           HEATER_ON => "DB2040_WINCC_HMI_LINES".SERVICES[9].WINCC_LINE_REQUEST_RIGHT,
                           DISC_SPEED_WARN_UP_LIMIT => "DB21003_POWDER_FEEDER_HMI_INTERLOCK".POWDER_FEEDER_2_UNIT_02."HMI_Offsets Alarms and Warnings".DiskSpeedNominalLine2_Max_Warning,
                           DISC_SPEED_ALRM_UP_LIMIT => "DB21003_POWDER_FEEDER_HMI_INTERLOCK".POWDER_FEEDER_2_UNIT_02."HMI_Offsets Alarms and Warnings".DiskSpeedNominalLine2_Max_Alarm,
                           DISC_SPEED_WARN_LOW_LIMIT => "DB21003_POWDER_FEEDER_HMI_INTERLOCK".POWDER_FEEDER_2_UNIT_02."HMI_Offsets Alarms and Warnings".DiskSpeedNominalLine2_Min_Warning,
                           DISC_SPEED_ALRM_LOW_LIMIT => "DB21003_POWDER_FEEDER_HMI_INTERLOCK".POWDER_FEEDER_2_UNIT_02."HMI_Offsets Alarms and Warnings".DiskSpeedNominalLine2_Min_Alarm,
                           GAS_FLOW_RATE_WARN_UP_LIMIT => "DB21003_POWDER_FEEDER_HMI_INTERLOCK".POWDER_FEEDER_2_UNIT_02."HMI_Offsets Alarms and Warnings".CarrierGasNominalLine2_Max_Warning,
                           GAS_FLOW_RATE_ALRM_UP_LIMIT => "DB21003_POWDER_FEEDER_HMI_INTERLOCK".POWDER_FEEDER_2_UNIT_02."HMI_Offsets Alarms and Warnings".CarrierGasNominalLine2_Max_Alarm,
                           GAS_FLOW_RATE_WARN_LOW_LIMIT => "DB21003_POWDER_FEEDER_HMI_INTERLOCK".POWDER_FEEDER_2_UNIT_02."HMI_Offsets Alarms and Warnings".CarrierGasNominalLine2_Min_Warning,
                           GAS_FLOW_RATE_ALRM_LOW_LIMIT => "DB21003_POWDER_FEEDER_HMI_INTERLOCK".POWDER_FEEDER_2_UNIT_02."HMI_Offsets Alarms and Warnings".CarrierGasNominalLine2_Min_Alarm,
                           STIRRER_SPEED_WARN_UP_LIMIT => "DB21003_POWDER_FEEDER_HMI_INTERLOCK".POWDER_FEEDER_2_UNIT_02."HMI_Offsets Alarms and Warnings".StirrerSpeedNominalLine2_Max_Warning,
                           STIRRER_SPEED_ALRM_UP_LIMIT => "DB21003_POWDER_FEEDER_HMI_INTERLOCK".POWDER_FEEDER_2_UNIT_02."HMI_Offsets Alarms and Warnings".StirrerSpeedNominalLine2_Max_Alarm,
                           STIRRER_SPEED_WARN_LOW_LIMIT => "DB21003_POWDER_FEEDER_HMI_INTERLOCK".POWDER_FEEDER_2_UNIT_02."HMI_Offsets Alarms and Warnings".StirrerSpeedNominalLine2_Min_Warning,
                           STIRRER_SPEED_ALRM_LOW_LIMIT => "DB21003_POWDER_FEEDER_HMI_INTERLOCK".POWDER_FEEDER_2_UNIT_02."HMI_Offsets Alarms and Warnings".StirrerSpeedNominalLine2_Min_Alarm,
                           TEMP_ALRM_UP_LIMIT => "DB21003_POWDER_FEEDER_HMI_INTERLOCK".POWDER_FEEDER_2_UNIT_02."HMI_Offsets Alarms and Warnings".HopperTempNominalLine2_Max_Alarm,
                           HOPPER_TEMP_MANUAL => "DB21003_POWDER_FEEDER_HMI_INTERLOCK".POWDER_FEEDER_2_UNIT_02."HMI_Values Setpoints".HopperTempNominalLine2,
                           STIRRER_SPEED_MANUAL => "DB21003_POWDER_FEEDER_HMI_INTERLOCK".POWDER_FEEDER_2_UNIT_02."HMI_Values Setpoints".StirrerSpeedNominalLine2,
                           DISC_SPEED_MANUAL => "DB21003_POWDER_FEEDER_HMI_INTERLOCK".POWDER_FEEDER_2_UNIT_02."HMI_Values Setpoints".DiskSpeedNominalLine2,
                           GAS_FLOW_RATE_MANUAL => "DB21003_POWDER_FEEDER_HMI_INTERLOCK".POWDER_FEEDER_2_UNIT_02."HMI_Values Setpoints".CarrierGasNominalLine2,
                           START_SEQUENCE_GAS_STEPS => "DB21033_PF_2_HOPPERS_UNIT_02".SWITCH_ON_SEQUENCE_LINE_2.MAX_STEPS_GAS,
                           START_SEQUENCE_DISK_STEPS => "DB21033_PF_2_HOPPERS_UNIT_02".SWITCH_ON_SEQUENCE_LINE_2.MAX_STEPS_DISK,
                           STOP_SEQUENCE_GAS_STEPS => "DB21033_PF_2_HOPPERS_UNIT_02".SWITCH_OFF_SEQUENCE_LINE_2.MAX_STEPS_GAS,
                           STOP_SEQUENCE_DISK_STEP => "DB21033_PF_2_HOPPERS_UNIT_02".SWITCH_OFF_SEQUENCE_LINE_2.MAX_STEPS_DISK,
                           STOP_SEQUENCE_PAUSE_STEP => "DB21033_PF_2_HOPPERS_UNIT_02".SWITCH_OFF_SEQUENCE_LINE_2.GAS_WAIT_STEP,
                           SELECTED_ARGON_GAS => "DB21003_POWDER_FEEDER_HMI_INTERLOCK".POWDER_FEEDER_2_UNIT_02.HMI_ACTIONS_STATUS.SELECTED_ARGON_GAS,
                           SELECTED_NITROGEN_GAS => "DB21003_POWDER_FEEDER_HMI_INTERLOCK".POWDER_FEEDER_2_UNIT_02.HMI_ACTIONS_STATUS.SELECTED_NITROGEN_GAS,
                           SELECTED_HELIUM_GAS => "DB21003_POWDER_FEEDER_HMI_INTERLOCK".POWDER_FEEDER_2_UNIT_02.HMI_ACTIONS_STATUS.SELECTED_HELIUM_GAS,
                           SELECTED_ARGON30_GAS => "DB21003_POWDER_FEEDER_HMI_INTERLOCK".POWDER_FEEDER_2_UNIT_02.HMI_ACTIONS_STATUS.SELECTED_ARGON30_GAS);
END_REGION

REGION Network 7: HOPPER 1 UNIT 01
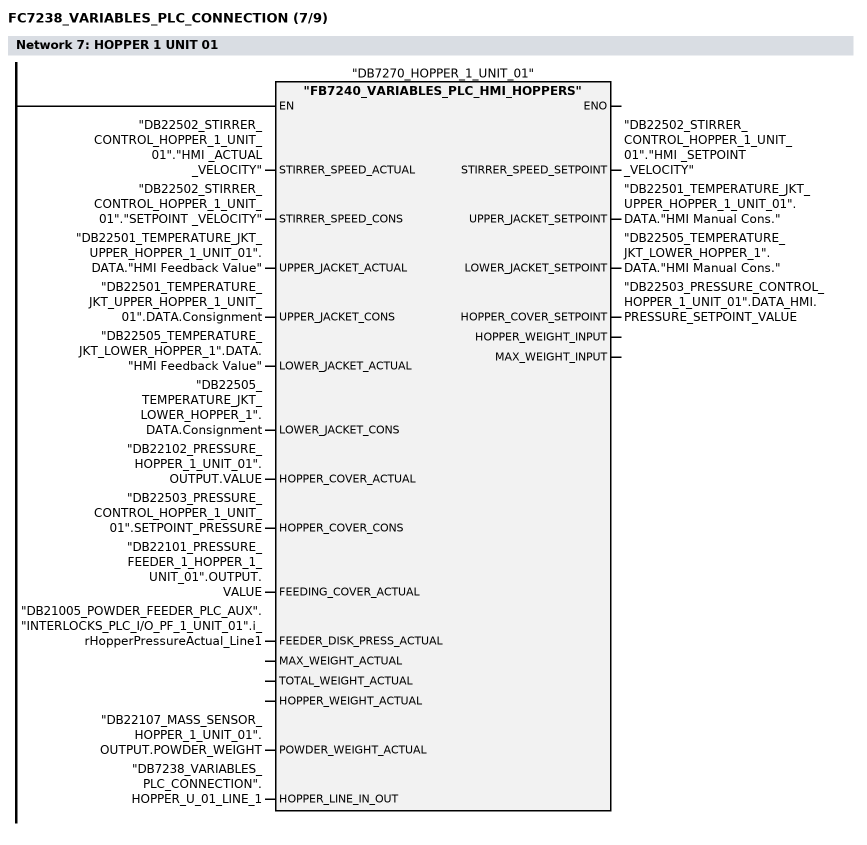
   RUNG wire#powerrail
      "DB7270_HOPPER_1_UNIT_01"(STIRRER_SPEED_ACTUAL := "DB22502_STIRRER_CONTROL_HOPPER_1_UNIT_01"."HMI _ACTUAL _VELOCITY", STIRRER_SPEED_CONS := "DB22502_STIRRER_CONTROL_HOPPER_1_UNIT_01"."SETPOINT _VELOCITY", UPPER_JACKET_ACTUAL := "DB22501_TEMPERATURE_JKT_UPPER_HOPPER_1_UNIT_01".DATA."HMI Feedback Value", UPPER_JACKET_CONS := "DB22501_TEMPERATURE_JKT_UPPER_HOPPER_1_UNIT_01".DATA.Consignment, LOWER_JACKET_ACTUAL := "DB22505_TEMPERATURE_JKT_LOWER_HOPPER_1".DATA."HMI Feedback Value", LOWER_JACKET_CONS := "DB22505_TEMPERATURE_JKT_LOWER_HOPPER_1".DATA.Consignment, HOPPER_COVER_ACTUAL := "DB22102_PRESSURE_HOPPER_1_UNIT_01".OUTPUT.VALUE, HOPPER_COVER_CONS := "DB22503_PRESSURE_CONTROL_HOPPER_1_UNIT_01".SETPOINT_PRESSURE, FEEDING_COVER_ACTUAL := "DB22101_PRESSURE_FEEDER_1_HOPPER_1_UNIT_01".OUTPUT.VALUE, FEEDER_DISK_PRESS_ACTUAL := "DB21005_POWDER_FEEDER_PLC_AUX"."INTERLOCKS_PLC_I/O_PF_1_UNIT_01".i_rHopperPressureActual_Line1, MAX_WEIGHT_ACTUAL :=, TOTAL_WEIGHT_ACTUAL :=, HOPPER_WEIGHT_ACTUAL :=, POWDER_WEIGHT_ACTUAL := "DB22107_MASS_SENSOR_HOPPER_1_UNIT_01".OUTPUT.POWDER_WEIGHT, HOPPER_LINE_IN_OUT := "DB7238_VARIABLES_PLC_CONNECTION".HOPPER_U_01_LINE_1, STIRRER_SPEED_SETPOINT => "DB22502_STIRRER_CONTROL_HOPPER_1_UNIT_01"."HMI _SETPOINT _VELOCITY", UPPER_JACKET_SETPOINT => "DB22501_TEMPERATURE_JKT_UPPER_HOPPER_1_UNIT_01".DATA."HMI Manual Cons.", LOWER_JACKET_SETPOINT => "DB22505_TEMPERATURE_JKT_LOWER_HOPPER_1".DATA."HMI Manual Cons.", HOPPER_COVER_SETPOINT => "DB22503_PRESSURE_CONTROL_HOPPER_1_UNIT_01".DATA_HMI.PRESSURE_SETPOINT_VALUE, HOPPER_WEIGHT_INPUT =>, MAX_WEIGHT_INPUT =>)
   END_RUNG
   // the same network as SCL:
   "DB7270_HOPPER_1_UNIT_01"(STIRRER_SPEED_ACTUAL := "DB22502_STIRRER_CONTROL_HOPPER_1_UNIT_01"."HMI _ACTUAL _VELOCITY",   // "FB7240_VARIABLES_PLC_HMI_HOPPERS"
                           STIRRER_SPEED_CONS := "DB22502_STIRRER_CONTROL_HOPPER_1_UNIT_01"."SETPOINT _VELOCITY",
                           UPPER_JACKET_ACTUAL := "DB22501_TEMPERATURE_JKT_UPPER_HOPPER_1_UNIT_01".DATA."HMI Feedback Value",
                           UPPER_JACKET_CONS := "DB22501_TEMPERATURE_JKT_UPPER_HOPPER_1_UNIT_01".DATA.Consignment,
                           LOWER_JACKET_ACTUAL := "DB22505_TEMPERATURE_JKT_LOWER_HOPPER_1".DATA."HMI Feedback Value",
                           LOWER_JACKET_CONS := "DB22505_TEMPERATURE_JKT_LOWER_HOPPER_1".DATA.Consignment,
                           HOPPER_COVER_ACTUAL := "DB22102_PRESSURE_HOPPER_1_UNIT_01".OUTPUT.VALUE,
                           HOPPER_COVER_CONS := "DB22503_PRESSURE_CONTROL_HOPPER_1_UNIT_01".SETPOINT_PRESSURE,
                           FEEDING_COVER_ACTUAL := "DB22101_PRESSURE_FEEDER_1_HOPPER_1_UNIT_01".OUTPUT.VALUE,
                           FEEDER_DISK_PRESS_ACTUAL := "DB21005_POWDER_FEEDER_PLC_AUX"."INTERLOCKS_PLC_I/O_PF_1_UNIT_01".i_rHopperPressureActual_Line1,
                           POWDER_WEIGHT_ACTUAL := "DB22107_MASS_SENSOR_HOPPER_1_UNIT_01".OUTPUT.POWDER_WEIGHT,
                           HOPPER_LINE_IN_OUT := "DB7238_VARIABLES_PLC_CONNECTION".HOPPER_U_01_LINE_1,
                           STIRRER_SPEED_SETPOINT => "DB22502_STIRRER_CONTROL_HOPPER_1_UNIT_01"."HMI _SETPOINT _VELOCITY",
                           UPPER_JACKET_SETPOINT => "DB22501_TEMPERATURE_JKT_UPPER_HOPPER_1_UNIT_01".DATA."HMI Manual Cons.",
                           LOWER_JACKET_SETPOINT => "DB22505_TEMPERATURE_JKT_LOWER_HOPPER_1".DATA."HMI Manual Cons.",
                           HOPPER_COVER_SETPOINT => "DB22503_PRESSURE_CONTROL_HOPPER_1_UNIT_01".DATA_HMI.PRESSURE_SETPOINT_VALUE);
END_REGION

REGION Network 8: EKS VALUES TO HMI
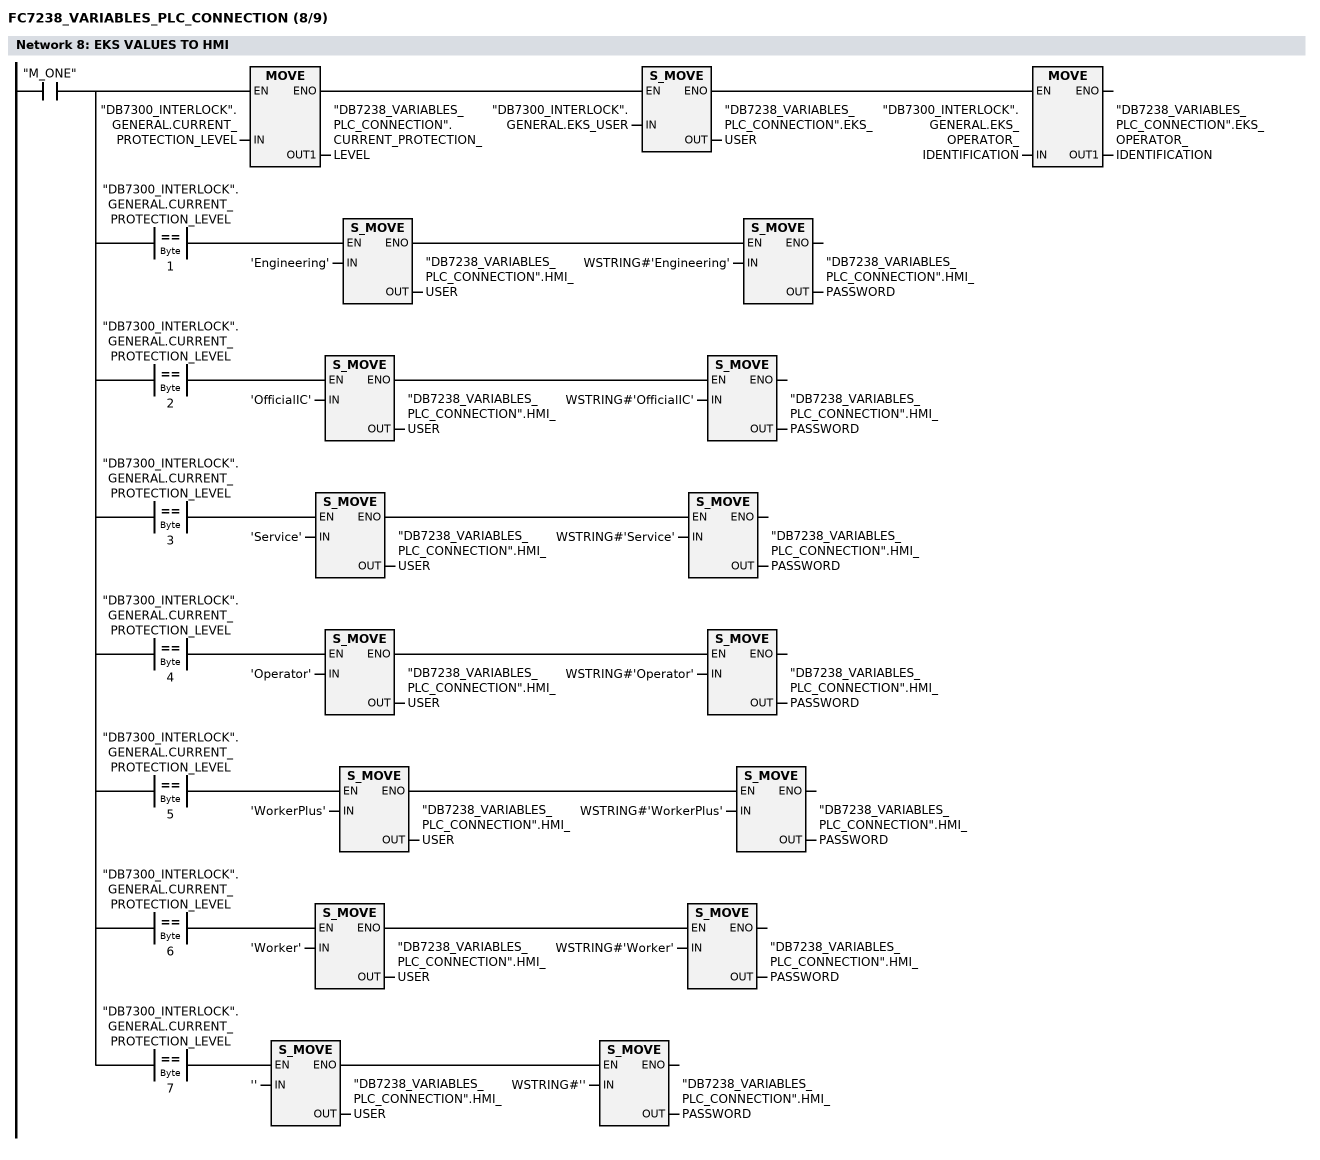
   RUNG wire#powerrail
      Contact( "M_ONE" )
      wire#w1
      Move(in := "DB7300_INTERLOCK".GENERAL.CURRENT_PROTECTION_LEVEL, out1 => "DB7238_VARIABLES_PLC_CONNECTION".CURRENT_PROTECTION_LEVEL)
      S_Move(in := "DB7300_INTERLOCK".GENERAL.EKS_USER, out => "DB7238_VARIABLES_PLC_CONNECTION".EKS_USER)
      Move(in := "DB7300_INTERLOCK".GENERAL.EKS_OPERATOR_IDENTIFICATION, out1 => "DB7238_VARIABLES_PLC_CONNECTION".EKS_OPERATOR_IDENTIFICATION)
   END_RUNG
   RUNG wire#w1
      { S7_Templates := "SrcType := Byte" } EQ_Contact(in1 := "DB7300_INTERLOCK".GENERAL.CURRENT_PROTECTION_LEVEL, in2 := 1)
      S_Move(in := 'Engineering', out => "DB7238_VARIABLES_PLC_CONNECTION".HMI_USER)
      S_Move(in := WSTRING#'Engineering', out => "DB7238_VARIABLES_PLC_CONNECTION".HMI_PASSWORD)
   END_RUNG
   RUNG wire#w1
      { S7_Templates := "SrcType := Byte" } EQ_Contact(in1 := "DB7300_INTERLOCK".GENERAL.CURRENT_PROTECTION_LEVEL, in2 := 2)
      S_Move(in := 'OfficialIC', out => "DB7238_VARIABLES_PLC_CONNECTION".HMI_USER)
      S_Move(in := WSTRING#'OfficialIC', out => "DB7238_VARIABLES_PLC_CONNECTION".HMI_PASSWORD)
   END_RUNG
   RUNG wire#w1
      { S7_Templates := "SrcType := Byte" } EQ_Contact(in1 := "DB7300_INTERLOCK".GENERAL.CURRENT_PROTECTION_LEVEL, in2 := 3)
      S_Move(in := 'Service', out => "DB7238_VARIABLES_PLC_CONNECTION".HMI_USER)
      S_Move(in := WSTRING#'Service', out => "DB7238_VARIABLES_PLC_CONNECTION".HMI_PASSWORD)
   END_RUNG
   RUNG wire#w1
      { S7_Templates := "SrcType := Byte" } EQ_Contact(in1 := "DB7300_INTERLOCK".GENERAL.CURRENT_PROTECTION_LEVEL, in2 := 4)
      S_Move(in := 'Operator', out => "DB7238_VARIABLES_PLC_CONNECTION".HMI_USER)
      S_Move(in := WSTRING#'Operator', out => "DB7238_VARIABLES_PLC_CONNECTION".HMI_PASSWORD)
   END_RUNG
   RUNG wire#w1
      { S7_Templates := "SrcType := Byte" } EQ_Contact(in1 := "DB7300_INTERLOCK".GENERAL.CURRENT_PROTECTION_LEVEL, in2 := 5)
      S_Move(in := 'WorkerPlus', out => "DB7238_VARIABLES_PLC_CONNECTION".HMI_USER)
      S_Move(in := WSTRING#'WorkerPlus', out => "DB7238_VARIABLES_PLC_CONNECTION".HMI_PASSWORD)
   END_RUNG
   RUNG wire#w1
      { S7_Templates := "SrcType := Byte" } EQ_Contact(in1 := "DB7300_INTERLOCK".GENERAL.CURRENT_PROTECTION_LEVEL, in2 := 6)
      S_Move(in := 'Worker', out => "DB7238_VARIABLES_PLC_CONNECTION".HMI_USER)
      S_Move(in := WSTRING#'Worker', out => "DB7238_VARIABLES_PLC_CONNECTION".HMI_PASSWORD)
   END_RUNG
   RUNG wire#w1
      { S7_Templates := "SrcType := Byte" } EQ_Contact(in1 := "DB7300_INTERLOCK".GENERAL.CURRENT_PROTECTION_LEVEL, in2 := 7)
      S_Move(in := '', out => "DB7238_VARIABLES_PLC_CONNECTION".HMI_USER)
      S_Move(in := WSTRING#'', out => "DB7238_VARIABLES_PLC_CONNECTION".HMI_PASSWORD)
   END_RUNG
   // the same network as SCL:
   IF "M_ONE" THEN
       "DB7238_VARIABLES_PLC_CONNECTION".CURRENT_PROTECTION_LEVEL := "DB7300_INTERLOCK".GENERAL.CURRENT_PROTECTION_LEVEL;
       "DB7238_VARIABLES_PLC_CONNECTION".EKS_USER := "DB7300_INTERLOCK".GENERAL.EKS_USER;
       "DB7238_VARIABLES_PLC_CONNECTION".EKS_OPERATOR_IDENTIFICATION := "DB7300_INTERLOCK".GENERAL.EKS_OPERATOR_IDENTIFICATION;
   END_IF;
   IF "M_ONE" AND ("DB7300_INTERLOCK".GENERAL.CURRENT_PROTECTION_LEVEL = 1) THEN
       "DB7238_VARIABLES_PLC_CONNECTION".HMI_USER := 'Engineering';
       "DB7238_VARIABLES_PLC_CONNECTION".HMI_PASSWORD := WSTRING#'Engineering';
   END_IF;
   IF "M_ONE" AND ("DB7300_INTERLOCK".GENERAL.CURRENT_PROTECTION_LEVEL = 2) THEN
       "DB7238_VARIABLES_PLC_CONNECTION".HMI_USER := 'OfficialIC';
       "DB7238_VARIABLES_PLC_CONNECTION".HMI_PASSWORD := WSTRING#'OfficialIC';
   END_IF;
   IF "M_ONE" AND ("DB7300_INTERLOCK".GENERAL.CURRENT_PROTECTION_LEVEL = 3) THEN
       "DB7238_VARIABLES_PLC_CONNECTION".HMI_USER := 'Service';
       "DB7238_VARIABLES_PLC_CONNECTION".HMI_PASSWORD := WSTRING#'Service';
   END_IF;
   IF "M_ONE" AND ("DB7300_INTERLOCK".GENERAL.CURRENT_PROTECTION_LEVEL = 4) THEN
       "DB7238_VARIABLES_PLC_CONNECTION".HMI_USER := 'Operator';
       "DB7238_VARIABLES_PLC_CONNECTION".HMI_PASSWORD := WSTRING#'Operator';
   END_IF;
   IF "M_ONE" AND ("DB7300_INTERLOCK".GENERAL.CURRENT_PROTECTION_LEVEL = 5) THEN
       "DB7238_VARIABLES_PLC_CONNECTION".HMI_USER := 'WorkerPlus';
       "DB7238_VARIABLES_PLC_CONNECTION".HMI_PASSWORD := WSTRING#'WorkerPlus';
   END_IF;
   IF "M_ONE" AND ("DB7300_INTERLOCK".GENERAL.CURRENT_PROTECTION_LEVEL = 6) THEN
       "DB7238_VARIABLES_PLC_CONNECTION".HMI_USER := 'Worker';
       "DB7238_VARIABLES_PLC_CONNECTION".HMI_PASSWORD := WSTRING#'Worker';
   END_IF;
   IF "M_ONE" AND ("DB7300_INTERLOCK".GENERAL.CURRENT_PROTECTION_LEVEL = 7) THEN
       "DB7238_VARIABLES_PLC_CONNECTION".HMI_USER := '';
       "DB7238_VARIABLES_PLC_CONNECTION".HMI_PASSWORD := WSTRING#'';
   END_IF;
END_REGION

REGION Network 9: GENERAL HMI PLC CONNECTION
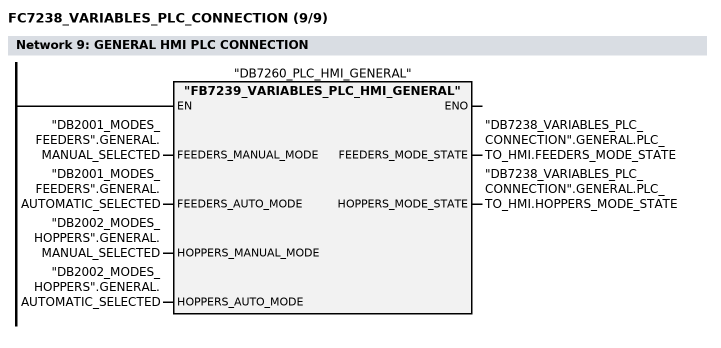
   RUNG wire#powerrail
      "DB7260_PLC_HMI_GENERAL"(FEEDERS_MANUAL_MODE := "DB2001_MODES_FEEDERS".GENERAL.MANUAL_SELECTED, FEEDERS_AUTO_MODE := "DB2001_MODES_FEEDERS".GENERAL.AUTOMATIC_SELECTED, HOPPERS_MANUAL_MODE := "DB2002_MODES_HOPPERS".GENERAL.MANUAL_SELECTED, HOPPERS_AUTO_MODE := "DB2002_MODES_HOPPERS".GENERAL.AUTOMATIC_SELECTED, FEEDERS_MODE_STATE => "DB7238_VARIABLES_PLC_CONNECTION".GENERAL.PLC_TO_HMI.FEEDERS_MODE_STATE, HOPPERS_MODE_STATE => "DB7238_VARIABLES_PLC_CONNECTION".GENERAL.PLC_TO_HMI.HOPPERS_MODE_STATE)
   END_RUNG
   // the same network as SCL:
   "DB7260_PLC_HMI_GENERAL"(FEEDERS_MANUAL_MODE := "DB2001_MODES_FEEDERS".GENERAL.MANUAL_SELECTED,   // "FB7239_VARIABLES_PLC_HMI_GENERAL"
                           FEEDERS_AUTO_MODE := "DB2001_MODES_FEEDERS".GENERAL.AUTOMATIC_SELECTED,
                           HOPPERS_MANUAL_MODE := "DB2002_MODES_HOPPERS".GENERAL.MANUAL_SELECTED,
                           HOPPERS_AUTO_MODE := "DB2002_MODES_HOPPERS".GENERAL.AUTOMATIC_SELECTED,
                           FEEDERS_MODE_STATE => "DB7238_VARIABLES_PLC_CONNECTION".GENERAL.PLC_TO_HMI.FEEDERS_MODE_STATE,
                           HOPPERS_MODE_STATE => "DB7238_VARIABLES_PLC_CONNECTION".GENERAL.PLC_TO_HMI.HOPPERS_MODE_STATE);
END_REGION
END_FUNCTION
